(*Przepisanie wystąpienia warningów*)
VIS.uliWarningOccure.0:= TanksWarning[0].bWarning; 			AudiActiveWarningDescriptionIDtemp[0] := 25;
VIS.uliWarningOccure.1:= TanksWarning[1].bWarning; 			AudiActiveWarningDescriptionIDtemp[1] := 26;
VIS.uliWarningOccure.2:= BottleTransferWarning[0].bWarning; AudiActiveWarningDescriptionIDtemp[2] := 57;
VIS.uliWarningOccure.3:= GeneralWarning1[0].bWarning;		AudiActiveWarningDescriptionIDtemp[3] := 65;
VIS.uliWarningOccure.4:= WeightWarning[0].bWarning;	AudiActiveWarningDescriptionIDtemp[4] := 73;
VIS.uliWarningOccure.5:= BottleTransferWarning[1].bWarning;	AudiActiveWarningDescriptionIDtemp[5] := 58;
VIS.uliWarningOccure.6:= GeneralWarning1[0].bWarning;	AudiActiveWarningDescriptionIDtemp[6] := 65;
VIS.uliWarningOccure.7:= GeneralWarning1[1].bWarning;	AudiActiveWarningDescriptionIDtemp[7] := 66;
VIS.uliWarningOccure.8:= GeneralWarning1[2].bWarning;	AudiActiveWarningDescriptionIDtemp[8] := 67;
VIS.uliWarningOccure.9:= GeneralWarning1[3].bWarning;	AudiActiveWarningDescriptionIDtemp[9] := 68;
VIS.uliWarningOccure.10:=DispencersWarning[0].bWarning;	AudiActiveWarningDescriptionIDtemp[10] := 17;
VIS.uliWarningOccure.11:=DispencersWarning[1].bWarning;	AudiActiveWarningDescriptionIDtemp[11] := 18;
VIS.uliWarningOccure.12:=DispencersWarning[2].bWarning;	AudiActiveWarningDescriptionIDtemp[12] := 19;
VIS.uliWarningOccure.13:=DispencersWarning[3].bWarning;	AudiActiveWarningDescriptionIDtemp[13] := 20;
VIS.uliWarningOccure.14:=DispencersWarning[4].bWarning;	AudiActiveWarningDescriptionIDtemp[14] := 21;
VIS.uliWarningOccure.15:=ScrewersWarning[0].bWarning; 	AudiActiveWarningDescriptionIDtemp[15] := 49;
VIS.uliWarningOccure.16:=ScrewersWarning[1].bWarning;	AudiActiveWarningDescriptionIDtemp[16] := 50;
VIS.uliWarningOccure.17:=ScrewersWarning[2].bWarning;	AudiActiveWarningDescriptionIDtemp[17] := 51;
VIS.uliWarningOccure.18:=ScrewersWarning[3].bWarning;	AudiActiveWarningDescriptionIDtemp[18] := 52;
VIS.uliWarningOccure.19:=ScrewersWarning[4].bWarning;	AudiActiveWarningDescriptionIDtemp[19] := 53;
VIS.uliWarningOccure.20:=ScrewersWarning[5].bWarning;	AudiActiveWarningDescriptionIDtemp[20] := 54;
VIS.uliWarningOccure.21:=ScrewersWarning[6].bWarning;	AudiActiveWarningDescriptionIDtemp[21] := 55;
VIS.uliWarningOccure.22:=ScrewersWarning[7].bWarning;	AudiActiveWarningDescriptionIDtemp[22] := 56;
VIS.uliWarningOccure.23:=BottleFeederWarning[0].bWarning; 	AudiActiveWarningDescriptionIDtemp[23] := 1;
VIS.uliWarningOccure.24:=ExSensorWarning[1].bWarning;	AudiActiveWarningDescriptionIDtemp[24] := 90;
VIS.uliWarningOccure.25:=CapFeederWarning[0].bWarning;	AudiActiveWarningDescriptionIDtemp[25] := 33;
VIS.uliWarningOccure.26:=BottleFeederWarning[1].bWarning;	AudiActiveWarningDescriptionIDtemp[26] := 2;

VIS.uliWarningOccure.41:=BottleFeederWarning[2].bWarning;	AudiActiveWarningDescriptionIDtemp[41] := 3;
VIS.uliWarningOccure.42:=BottleFeederWarning[3].bWarning;	AudiActiveWarningDescriptionIDtemp[42] := 4;

VIS.uliWarningOccure.27:=CapSorterWarning[0].bWarning;	AudiActiveWarningDescriptionIDtemp[27] := 41;
VIS.uliWarningOccure.28:=CapSorterWarning[1].bWarning;	AudiActiveWarningDescriptionIDtemp[28] := 42;
VIS.uliWarningOccure.29:=CapSorterWarning[2].bWarning;	AudiActiveWarningDescriptionIDtemp[29] := 43;
VIS.uliWarningOccure.30:=CapSorterWarning[3].bWarning;	AudiActiveWarningDescriptionIDtemp[30] := 44;
VIS.uliWarningOccure.31:=CapSorterWarning[4].bWarning;	AudiActiveWarningDescriptionIDtemp[31] := 45;
VIS.uliWarningOccure.32:=CapSorterWarning[5].bWarning;	AudiActiveWarningDescriptionIDtemp[32] := 46;

VIS.uliWarningOccure.33:=BottleSorterWarning[0].bWarning;	AudiActiveWarningDescriptionIDtemp[33] := 9;
VIS.uliWarningOccure.34:=BottleSorterWarning[1].bWarning;	AudiActiveWarningDescriptionIDtemp[34] := 10;
VIS.uliWarningOccure.35:=BottleSorterWarning[2].bWarning;	AudiActiveWarningDescriptionIDtemp[35] := 11;
VIS.uliWarningOccure.36:=BottleSorterWarning[3].bWarning;	AudiActiveWarningDescriptionIDtemp[36] := 12;
VIS.uliWarningOccure.37:=BottleSorterWarning[4].bWarning;	AudiActiveWarningDescriptionIDtemp[37] := 13;
VIS.uliWarningOccure.38:=BottleSorterWarning[5].bWarning;	AudiActiveWarningDescriptionIDtemp[48] := 14;

VIS.uliWarningOccure.39:=LidFeederWarning[0].bWarning;	AudiActiveWarningDescriptionIDtemp[39] := 		81;
VIS.uliWarningOccure.40:=LidFeederWarning[1].bWarning;	AudiActiveWarningDescriptionIDtemp[40] := 		82;

(*Potwierdź wszystkie ostrzeżenia*)
IF VIS.bWarningAcknowledgeAll THEN
	VIS.uliWarningAcknowledge	:=	2#111111111111111111111111111111111111111111111111111111111;
	VIS.bWarningAcknowledgeAll	:= 	FALSE;
	iWarningAcknowledgeAll		:=	iWarningAcknowledgeAll	+	1;  // Sprawdzanie ile razy było wciśnięte
END_IF

(*Potwierdzenia*)
IF VIS.uliWarningAcknowledge.0 THEN TanksWarning[0].bAcknowledge					:=TRUE;	END_IF
IF VIS.uliWarningAcknowledge.1 THEN TanksWarning[1].bAcknowledge					:=TRUE; END_IF
IF VIS.uliWarningAcknowledge.2 THEN BottleTransferWarning[0].bAcknowledge			:=TRUE; END_IF
IF VIS.uliWarningAcknowledge.3 THEN GeneralWarning1[0].bAcknowledge					:=TRUE; END_IF
IF VIS.uliWarningAcknowledge.4 THEN WeightWarning[0].bAcknowledge					:=TRUE; END_IF
IF VIS.bBottleTransferLubricationReset THEN BottleTransferWarning[1].bAcknowledge	:=TRUE; END_IF
IF VIS.uliWarningAcknowledge.6 THEN GeneralWarning1[1].bAcknowledge					:=TRUE; END_IF
IF VIS.uliWarningAcknowledge.7 THEN GeneralWarning1[2].bAcknowledge					:=TRUE; END_IF
IF VIS.uliWarningAcknowledge.8 THEN GeneralWarning1[3].bAcknowledge					:=TRUE; END_IF
IF VIS.uliWarningAcknowledge.9 THEN GeneralWarning1[4].bAcknowledge					:=TRUE; END_IF
IF VIS.uliWarningAcknowledge.10 THEN DispencersWarning[0].bAcknowledge				:=TRUE; END_IF
IF VIS.uliWarningAcknowledge.11 THEN DispencersWarning[1].bAcknowledge				:=TRUE; END_IF
IF VIS.uliWarningAcknowledge.12 THEN DispencersWarning[2].bAcknowledge				:=TRUE; END_IF
IF VIS.uliWarningAcknowledge.13 THEN DispencersWarning[3].bAcknowledge				:=TRUE; END_IF
IF VIS.uliWarningAcknowledge.14 THEN DispencersWarning[4].bAcknowledge				:=TRUE; END_IF
IF VIS.uliWarningAcknowledge.15 THEN ScrewersWarning[0].bAcknowledge				:=TRUE; END_IF
IF VIS.uliWarningAcknowledge.16 THEN ScrewersWarning[1].bAcknowledge				:=TRUE; END_IF
IF VIS.uliWarningAcknowledge.17 THEN ScrewersWarning[2].bAcknowledge				:=TRUE; END_IF
IF VIS.uliWarningAcknowledge.18 THEN ScrewersWarning[3].bAcknowledge				:=TRUE; END_IF
IF VIS.uliWarningAcknowledge.19 THEN ScrewersWarning[4].bAcknowledge				:=TRUE; END_IF
IF VIS.uliWarningAcknowledge.20 THEN ScrewersWarning[5].bAcknowledge				:=TRUE; END_IF
IF VIS.uliWarningAcknowledge.21 THEN ScrewersWarning[6].bAcknowledge				:=TRUE; END_IF
IF VIS.uliWarningAcknowledge.22 THEN ScrewersWarning[7].bAcknowledge				:=TRUE; END_IF
IF VIS.uliWarningAcknowledge.23 THEN BottleFeederWarning[0].bAcknowledge			:=TRUE; END_IF
IF VIS.uliWarningAcknowledge.24 THEN ExSensorWarning[1].bAcknowledge				:=TRUE; END_IF
IF VIS.uliWarningAcknowledge.25 THEN CapFeederWarning[0].bAcknowledge				:=TRUE; END_IF
IF VIS.uliWarningAcknowledge.26 THEN BottleFeederWarning[1].bAcknowledge			:=TRUE; END_IF	

IF VIS.uliWarningAcknowledge.41 THEN BottleFeederWarning[2].bAcknowledge			:=TRUE; END_IF	
IF VIS.uliWarningAcknowledge.42 THEN BottleFeederWarning[3].bAcknowledge			:=TRUE; END_IF	

IF VIS.uliWarningAcknowledge.27 THEN CapSorterWarning[0].bAcknowledge				:=TRUE; END_IF	
IF VIS.uliWarningAcknowledge.28 THEN CapSorterWarning[1].bAcknowledge				:=TRUE; END_IF
IF VIS.uliWarningAcknowledge.29 THEN CapSorterWarning[2].bAcknowledge				:=TRUE; END_IF
IF VIS.uliWarningAcknowledge.30 THEN CapSorterWarning[3].bAcknowledge				:=TRUE; END_IF
IF VIS.uliWarningAcknowledge.31 THEN CapSorterWarning[4].bAcknowledge				:=TRUE; END_IF
IF VIS.uliWarningAcknowledge.32 THEN CapSorterWarning[5].bAcknowledge				:=TRUE; END_IF

IF VIS.uliWarningAcknowledge.33 THEN BottleSorterWarning[0].bAcknowledge			:=TRUE; END_IF	
IF VIS.uliWarningAcknowledge.34 THEN BottleSorterWarning[1].bAcknowledge			:=TRUE; END_IF
IF VIS.uliWarningAcknowledge.35 THEN BottleSorterWarning[2].bAcknowledge			:=TRUE; END_IF
IF VIS.uliWarningAcknowledge.36 THEN BottleSorterWarning[3].bAcknowledge			:=TRUE; END_IF
IF VIS.uliWarningAcknowledge.37 THEN BottleSorterWarning[4].bAcknowledge			:=TRUE; END_IF
IF VIS.uliWarningAcknowledge.38 THEN BottleSorterWarning[5].bAcknowledge			:=TRUE; END_IF

IF VIS.uliWarningAcknowledge.39 THEN LidFeederWarning[0].bAcknowledge				:=TRUE; END_IF
IF VIS.uliWarningAcknowledge.40 THEN LidFeederWarning[1].bAcknowledge				:=TRUE; END_IF
//41 i 42 zajete

(*Opisy*)
VIS.AsWarningDescription[0]:=TanksWarning[0].sDescription;
VIS.AsWarningDescription[1]:=TanksWarning[1].sDescription;
VIS.AsWarningDescription[2]:=BottleTransferWarning[0].sDescription;
VIS.AsWarningDescription[3]:=GeneralWarning1[0].sDescription;
VIS.AsWarningDescription[4]:=WeightWarning[0].sDescription;
VIS.AsWarningDescription[5]:=BottleTransferWarning[1].sDescription;
VIS.AsWarningDescription[6]:=GeneralWarning1[1].sDescription;
VIS.AsWarningDescription[7]:=GeneralWarning1[2].sDescription;
VIS.AsWarningDescription[8]:=GeneralWarning1[3].sDescription;
VIS.AsWarningDescription[9]:=GeneralWarning1[4].sDescription;
VIS.AsWarningDescription[10]:=DispencersWarning[0].sDescription;
VIS.AsWarningDescription[11]:=DispencersWarning[1].sDescription;
VIS.AsWarningDescription[12]:=DispencersWarning[2].sDescription;
VIS.AsWarningDescription[13]:=DispencersWarning[3].sDescription;
VIS.AsWarningDescription[14]:=DispencersWarning[4].sDescription;
VIS.AsWarningDescription[15]:=ScrewersWarning[0].sDescription;
VIS.AsWarningDescription[16]:=ScrewersWarning[1].sDescription;
VIS.AsWarningDescription[17]:=ScrewersWarning[2].sDescription;
VIS.AsWarningDescription[18]:=ScrewersWarning[3].sDescription;
VIS.AsWarningDescription[19]:=ScrewersWarning[4].sDescription;
VIS.AsWarningDescription[20]:=ScrewersWarning[5].sDescription;
VIS.AsWarningDescription[21]:=ScrewersWarning[6].sDescription;
VIS.AsWarningDescription[22]:=ScrewersWarning[7].sDescription;
VIS.AsWarningDescription[23]:=BottleFeederWarning[0].sDescription;     
VIS.AsWarningDescription[24]:=ExSensorWarning[1].sDescription;
VIS.AsWarningDescription[25]:=CapFeederWarning[0].sDescription;
VIS.AsWarningDescription[26]:=BottleFeederWarning[1].sDescription;

VIS.AsWarningDescription[41]:=BottleFeederWarning[2].sDescription;
VIS.AsWarningDescription[42]:=BottleFeederWarning[3].sDescription;

VIS.AsWarningDescription[27]:=CapSorterWarning[0].sDescription;
VIS.AsWarningDescription[28]:=CapSorterWarning[1].sDescription;
VIS.AsWarningDescription[29]:=CapSorterWarning[2].sDescription;
VIS.AsWarningDescription[30]:=CapSorterWarning[3].sDescription;
VIS.AsWarningDescription[31]:=CapSorterWarning[4].sDescription;
VIS.AsWarningDescription[32]:=CapSorterWarning[5].sDescription;

VIS.AsWarningDescription[33]:=BottleSorterWarning[0].sDescription;
VIS.AsWarningDescription[34]:=BottleSorterWarning[1].sDescription;
VIS.AsWarningDescription[35]:=BottleSorterWarning[2].sDescription;
VIS.AsWarningDescription[36]:=BottleSorterWarning[3].sDescription;
VIS.AsWarningDescription[37]:=BottleSorterWarning[4].sDescription;
VIS.AsWarningDescription[38]:=BottleSorterWarning[5].sDescription;

VIS.AsWarningDescription[39]:=LidFeederWarning[0].sDescription;
VIS.AsWarningDescription[40]:=LidFeederWarning[1].sDescription;
//41 i 42 zajete


(*SYGNALIZOWANIE WARNINGOW*)
tonSoftAlarm(IN:=bSoftAlarm, PT:=T#500MS);
rtWarningOccure0(CLK:=VIS.uliWarningOccure.0,Q=>);
rtWarningOccure1(CLK:=VIS.uliWarningOccure.1,Q=>);
rtWarningOccure2(CLK:=VIS.uliWarningOccure.2,Q=>);
rtWarningOccure3(CLK:=VIS.uliWarningOccure.3,Q=>);
rtWarningOccure4(CLK:=VIS.uliWarningOccure.4,Q=>);
rtWarningOccure5(CLK:=VIS.uliWarningOccure.5,Q=>);
rtWarningOccure6(CLK:=VIS.uliWarningOccure.6,Q=>);
rtWarningOccure7(CLK:=VIS.uliWarningOccure.7,Q=>);
rtWarningOccure8(CLK:=VIS.uliWarningOccure.8,Q=>);
rtWarningOccure9(CLK:=VIS.uliWarningOccure.9,Q=>);
rtWarningOccure10(CLK:=VIS.uliWarningOccure.10,Q=>);
rtWarningOccure11(CLK:=VIS.uliWarningOccure.11,Q=>);
rtWarningOccure12(CLK:=VIS.uliWarningOccure.12,Q=>);
rtWarningOccure13(CLK:=VIS.uliWarningOccure.13,Q=>);
rtWarningOccure14(CLK:=VIS.uliWarningOccure.14,Q=>);
rtWarningOccure15(CLK:=VIS.uliWarningOccure.15,Q=>);
rtWarningOccure16(CLK:=VIS.uliWarningOccure.16,Q=>);
rtWarningOccure17(CLK:=VIS.uliWarningOccure.17,Q=>);
rtWarningOccure18(CLK:=VIS.uliWarningOccure.18,Q=>);
rtWarningOccure19(CLK:=VIS.uliWarningOccure.19,Q=>);
rtWarningOccure20(CLK:=VIS.uliWarningOccure.20,Q=>);
rtWarningOccure21(CLK:=VIS.uliWarningOccure.21,Q=>);
rtWarningOccure22(CLK:=VIS.uliWarningOccure.22,Q=>);
rtWarningOccure23(CLK:=VIS.uliWarningOccure.23,Q=>);
rtWarningOccure24(CLK:=VIS.uliWarningOccure.24,Q=>);
rtWarningOccure25(CLK:=VIS.uliWarningOccure.25,Q=>);
rtWarningOccure26(CLK:=VIS.uliWarningOccure.26,Q=>);

rtWarningOccure41(CLK:=VIS.uliWarningOccure.41,Q=>);
rtWarningOccure42(CLK:=VIS.uliWarningOccure.42,Q=>);

rtWarningOccure27(CLK:=VIS.uliWarningOccure.27,Q=>);
rtWarningOccure28(CLK:=VIS.uliWarningOccure.28,Q=>);
rtWarningOccure29(CLK:=VIS.uliWarningOccure.29,Q=>);
rtWarningOccure30(CLK:=VIS.uliWarningOccure.30,Q=>);
rtWarningOccure31(CLK:=VIS.uliWarningOccure.31,Q=>);
rtWarningOccure32(CLK:=VIS.uliWarningOccure.32,Q=>);

rtWarningOccure33(CLK:=VIS.uliWarningOccure.33,Q=>);
rtWarningOccure34(CLK:=VIS.uliWarningOccure.34,Q=>);
rtWarningOccure35(CLK:=VIS.uliWarningOccure.35,Q=>);
rtWarningOccure36(CLK:=VIS.uliWarningOccure.36,Q=>);
rtWarningOccure37(CLK:=VIS.uliWarningOccure.37,Q=>);
rtWarningOccure38(CLK:=VIS.uliWarningOccure.38,Q=>);

rtWarningOccure39(CLK:=VIS.uliWarningOccure.39,Q=>);
rtWarningOccure40(CLK:=VIS.uliWarningOccure.40,Q=>);

IF	(rtWarningOccure0.Q AND NOT VIS.uliWarningAcknowledge.0) OR
	(rtWarningOccure1.Q AND NOT VIS.uliWarningAcknowledge.1) OR
	(rtWarningOccure2.Q AND NOT VIS.uliWarningAcknowledge.2) OR
	(rtWarningOccure3.Q AND NOT VIS.uliWarningAcknowledge.3) OR
	(rtWarningOccure4.Q AND NOT VIS.uliWarningAcknowledge.4) OR
	(rtWarningOccure5.Q AND NOT VIS.uliWarningAcknowledge.5) OR
	(rtWarningOccure6.Q AND NOT VIS.uliWarningAcknowledge.6) OR	
	(rtWarningOccure7.Q AND NOT VIS.uliWarningAcknowledge.7) OR	
	(rtWarningOccure8.Q AND NOT VIS.uliWarningAcknowledge.8) OR	
	(rtWarningOccure9.Q AND NOT VIS.uliWarningAcknowledge.9) OR	
	(rtWarningOccure10.Q AND NOT VIS.uliWarningAcknowledge.10) OR	
	(rtWarningOccure11.Q AND NOT VIS.uliWarningAcknowledge.11) OR	
	(rtWarningOccure12.Q AND NOT VIS.uliWarningAcknowledge.12) OR	
	(rtWarningOccure13.Q AND NOT VIS.uliWarningAcknowledge.13) OR	
	(rtWarningOccure14.Q AND NOT VIS.uliWarningAcknowledge.14) OR	
	(rtWarningOccure15.Q AND NOT VIS.uliWarningAcknowledge.15) OR	
	(rtWarningOccure16.Q AND NOT VIS.uliWarningAcknowledge.16) OR	
	(rtWarningOccure17.Q AND NOT VIS.uliWarningAcknowledge.17) OR	
	(rtWarningOccure18.Q AND NOT VIS.uliWarningAcknowledge.18) OR	
	(rtWarningOccure19.Q AND NOT VIS.uliWarningAcknowledge.19) OR	
	(rtWarningOccure20.Q AND NOT VIS.uliWarningAcknowledge.20) OR	
	(rtWarningOccure21.Q AND NOT VIS.uliWarningAcknowledge.21) OR	
	(rtWarningOccure22.Q AND NOT VIS.uliWarningAcknowledge.22) OR
	(rtWarningOccure23.Q AND NOT VIS.uliWarningAcknowledge.23) OR
	(rtWarningOccure24.Q AND NOT VIS.uliWarningAcknowledge.24) OR
	(rtWarningOccure25.Q AND NOT VIS.uliWarningAcknowledge.25) OR
	(rtWarningOccure26.Q AND NOT VIS.uliWarningAcknowledge.26) OR
	(rtWarningOccure41.Q AND NOT VIS.uliWarningAcknowledge.41) OR
	(rtWarningOccure42.Q AND NOT VIS.uliWarningAcknowledge.42) OR
	(rtWarningOccure27.Q AND NOT VIS.uliWarningAcknowledge.27) OR
	(rtWarningOccure28.Q AND NOT VIS.uliWarningAcknowledge.28) OR
	(rtWarningOccure29.Q AND NOT VIS.uliWarningAcknowledge.29) OR
	(rtWarningOccure30.Q AND NOT VIS.uliWarningAcknowledge.30) OR
	(rtWarningOccure31.Q AND NOT VIS.uliWarningAcknowledge.31) OR
	(rtWarningOccure32.Q AND NOT VIS.uliWarningAcknowledge.32) OR
	(rtWarningOccure33.Q AND NOT VIS.uliWarningAcknowledge.33) OR
	(rtWarningOccure34.Q AND NOT VIS.uliWarningAcknowledge.34) OR
	(rtWarningOccure35.Q AND NOT VIS.uliWarningAcknowledge.35) OR
	(rtWarningOccure36.Q AND NOT VIS.uliWarningAcknowledge.36) OR
	(rtWarningOccure37.Q AND NOT VIS.uliWarningAcknowledge.37) OR
	(rtWarningOccure38.Q AND NOT VIS.uliWarningAcknowledge.38) OR
	(rtWarningOccure39.Q AND NOT VIS.uliWarningAcknowledge.39) OR
	(rtWarningOccure40.Q AND NOT VIS.uliWarningAcknowledge.40) 
	
	
 THEN
	bSoftAlarm:=TRUE;
END_IF
IF tonSoftAlarm.Q THEN
	bSoftAlarm:=FALSE;
END_IF


(*Wykrywanie nowego ostrzezenia do wizualizacji*)
rtWarningNew ( CLK:= uliWarningAcknowledgeTemp	<> VIS.uliWarningOccure AND VIS.uliWarningOccure > 0);
uliWarningAcknowledgeTemp	:=	VIS.uliWarningOccure;
IF rtWarningNew.Q THEN
	VIS.bWarningNew	:=	TRUE;
END_IF
tonWarningNew (IN:= VIS.bWarningNew ,PT:=T#1S);
IF tonWarningNew.Q THEN
	VIS.bWarningNew	:=	FALSE;
END_IF
(*Koniec Wykrywanie nowego ostrzezenia do wizualizacji*)
END_ACTION

END_PROGRAM

// ---- POUs/P11_RollerScrewer.TcPOU
(*
Nazwa:			P11_RollerScrewer
Opis:			Stacja zakręcarki rolkowej
Wersja:			v0.1
Data:			2018-10-10
Autor:			DP
Urzadzenia:		
Konfiguracja:	
Info:

*)
PROGRAM P11_RollerScrewer
VAR_INPUT

END_VAR
VAR
	(*********Zakręcarka rolkowa******)
	fbRollerScrewer: FB_RollerScrewer;		// Blok sterowania zakręcarką rolkową
	eRollerScrewerState: 			E_Station;						// Stan zakręcarki
	eRollerScrewerRunningState: 	E_RollerScrewer;				// Stan zakręcarki
	fbRollerScrewerState: 			FB_State;
	
	(************Chwytak*************)	
	fbRollerScrewerCatchStation						: FB_CatchStation;		
	eRollerScrewerCatchState						: E_Station;            
	eRollerScrewerCatchRunningState					: E_CatchStationState;  
	fbRollerScrewerCatchState						: FB_State;
	
	(************Szlaban*************)		
	fbRollerScrewerGate								: FB_SpringGateV2;

	
	// WEJŚĆIA I WYJŚCIA SPRZĘTOWE
	IbRollerScrewerHeightEncoderSetCDone			AT %I*: BOOL;
	IudiRollerScrewerHeightEncoderCV          		AT %I*: UDINT;
	QbRollerScrewerHeightEncoderSetC 				AT %Q*: BOOL;
	QudiRollerScrewerHeightEncoderSetCV       		AT %Q*: UDINT;

	QbRollerScrewerCatchHeightUpCmd 				AT %Q*: BOOL; 		
	QbRollerScrewerCatchHeightDownCmd 				AT %Q*: BOOL; 		
	IbRollerScrewerCatchHeightEncoderSetCDone		AT %I*: BOOL;
	IudiRollerScrewerCatchHeightEncoderCV          	AT %I*: UDINT;
	QbRollerScrewerCatchHeightEncoderSetC 			AT %Q*: BOOL;
	QudiRollerScrewerCatchHeightEncoderSetCV       	AT %Q*: UDINT;

	QABPneumaticRollerScrewerValveCoils 			AT %Q* 	: ARRAY[1..5] OF BYTE;	
	IuiPneumaticRollerScrewerState					AT %I* 	: UINT;	


	IbRollerScrewerFuseFB1OK						AT %I*	:BOOL;		
	IbRollerScrewerFuseRollerScrewerOK				AT %I*	:BOOL;		
	IbRollerScrewerFuseRollerScrewerCatchOK			AT %I*	:BOOL;		
	IbRollerScrewerPowerSupplyOK					AT %I*	:BOOL;
	//GVL_IO_SAFETY.IbSafetyRelayRC40	 			AT %I*  :BOOL;	
	IbRollerScrewerDoors1Open 						AT %I*	:BOOL;		
	IbRollerScrewerCycleStartStopButton				AT %I*	:BOOL;	
	IbRollerScrewerCompressedAirOK 					AT %I*	:BOOL;		
	IbRollerScrewerUnPressedTopSensor 				AT %I*	:BOOL;	
	IbRollerScrewerRollsUnPressedSensor 			AT %I*	:BOOL; 

	IbRollerScrewerCatchSensorOpened				AT %I*	:BOOL; 
	IbRollerScrewerDoors2Open 						AT %I*	:BOOL;			
	IbRollerScrewerCapPuttedSensor 					AT %I*	:BOOL;	
	QbRollerScrewerGreenSignalizationLamp 			AT %Q* : BOOL;			
	QbRollerScrewerRedSignalizationLamp 			AT %Q* : BOOL;				
	QbRollerScrewerWhiteSignalizationLamp 			AT %Q* : BOOL;						
	QbRollerScrewerYellowSignalizationLamp 			AT %Q* : BOOL;							
	QbRollerScrewerHeightMotorUp 					AT %Q*: BOOL;		
	QbRollerScrewerHeightMotorDown 					AT %Q*: BOOL;			
	
	QbRollerScrewerGate								: BOOL; 	
	QbRollerScrewerPressingTopActuator				: BOOL; 	
	QbRollerScrewerPressingRollsActuator			: BOOL; 	
	QbRollerScrewerCatchActuator					: BOOL; 

	QnRollerScrewerFrontTorqueLimit 				AT %Q*: UINT; 
	QnRollerScrewerRearTorqueLimit 					AT %Q*: UINT; 
	IrRollerScrewerRearActualMotorTemperature 		AT %I*: REAL; 
	IrRollerScrewerFrontActualMotorTemperature 		AT %I*: REAL; 

	(*RFID*)
	//Przed
	bReadedCard 										: BOOL;				
	nReadedCard											: ULINT;	
	fbReader   											: FB_IfmIoLinkRfid;
	AusiReaderInputData  								AT %I* : ARRAY[0..27] OF USINT;
	IbReaderTagPresent									AT %I* : BOOL;
	IBReaderErrorValue									AT %I* : BYTE;
	IbReaderCmdEnd										AT %I* : BOOL;
	IBReaderDataCounterIn								AT %I* : BYTE;
	IbReaderCmdStartAck									AT %I* : BOOL;
	IbReaderCmdStart									AT %Q* : BOOL;
	IBReaderCmmandValue									AT %Q* : BYTE;
	IBReaderDataCounterOut								AT %Q* : BYTE;
	AusiReaderOutputData  								AT %Q* : ARRAY[0..27] OF USINT;	


	TimerRollerScrewerEnable: TOF;
	TimerRollerScrewerCatchEnable: TOF;
	tonLidPuttedCheckEnable: TON;	
	rtEnable: R_TRIG;	
	
	(*Wykres dozowania*)
	fbRollerScrewingChart: FB_WriteDataToArrayString;

	rtStartRollerScrewing: R_TRIG;
	lrRollerScrewerAxisStartPosition: LREAL;

	tonRollerScrewerCatchSensorOpened: TON;
	


END_VAR

aPowerSupply();
aButtons();
aPneumatics();
aRFID();
aRFID_FB();
aSafety();
aSignalization();
aLimits();
a1_Gate();
a1_GateTime();
a2_RollerScrewer();
aWarnings();

(*** SKALOWANIE WARTOŚCI ZAKRĘCANIA Z Nm na % ***)
(* Wersja w Nm fbRollerScrewer.iScrewerSetTorque 
:=LREAL_TO_INT( 
													(lrRollerScrewingTightTorque/(INT_TO_LREAL(iPackageCapDiameter)*0.0633))*100
												 );*)
												 
fbRollerScrewer.iScrewerSetTorque :=LREAL_TO_INT(lrRollerScrewingTightTorque);												 
(*** KONIEC SKALOWANIE WARTOŚCI ZAKRĘCANIA Z Nm na % ***)

(*SYMULACJA CZUJNIKÓW*)
tonRollerScrewerCatchSensorOpened(IN:=NOT QbRollerScrewerCatchActuator, PT:=T#10MS);//bylo 300


(* BAZOWANIE - ZMIAN*)
tonLidPuttedCheckEnable(IN:=fbRollerScrewer.bEnable,PT:=T#5S); (*Dodany ton bo Wizka zjebnie wgrywa zmienne, najpierw włacza Enabla a potem dopiero wybiera recepture*)
//rtEnable(CLK:=fbRollerScrewer.bEnable,Q=>);
rtEnable(CLK:=tonLidPuttedCheckEnable.Q,Q=>);
// IF rtEnable.Q AND eMachineState>=E_MachineState.eReady AND eMachineState<>E_MachineState.eHardError  THEN
// 	VIS.bRollerScrewerCatchHeightSet:=TRUE;
// 	//VIS.bRollerScrewerHeightSet:=TRUE;
// ELSIF fbRollerScrewer.eState=E_Station.eHomingDone OR eMachineState=E_MachineState.eHardError THEN
//  	VIS.bRollerScrewerHeightSet:=FALSE;
// ELSIF  fbRollerScrewerCatchStation.eState=E_Station.eHomingDone OR eMachineState=E_MachineState.eHardError THEN
// 	VIS.bRollerScrewerHeightSet:=TRUE; //Zmiana LU208
// 	VIS.bRollerScrewerCatchHeightSet:=FALSE;
// END_IF
(*KONIEC BAZOWANIE - ZMIANA*)


(********* GENEROWANIE STANU STACJI DO WIZKI**********)
// fbRollerScrewerState(
// 	eState:=eRollerScrewerState , 
// 	bRun:=bStartRollerScrewing OR VIS.bManualStartRollerScrew,	
// 	eRollerScrewerRunningState:=eRollerScrewerRunningState , 
// 	sStateDesc=> VIS.sRollerScrewerState,
// 	iState=>VIS.iRollerScrewerState);
//fbRollerScrewerCatchState(
//	eState:=eRollerScrewerCatchState , 
//	bRun:=bRollerScrewerCatch,	
//	eCatchRunningState:=eRollerScrewerCatchRunningState , 
//	sStateDesc=> VIS.sRollerScrewerCatchState,
//	iState=>VIS.iRollerScrewerCatchState);	
(***** KONIEC GENEROWANIE STANU STACJI DO WIZKI*******)

(*Opoznienie wyłączanie enabla*)
TimerRollerScrewerEnable 		(IN:=bRollerScrewerEnable  AND NOT bChangeover , PT:=T#2S);
TimerRollerScrewerCatchEnable 	(IN:=bRollerScrewerEnable  AND NOT bChangeover , PT:=T#4S);
{warning 'Zmienione włączenie/wyłączanie rolkowej do testów'}

(*Przypisywanie wartości*)
IF fbRollerScrewerCatchStation.lrHeightMotorCV+24 <= 65 THEN //Warrtość minimalna stacji zakrecarki rolkowej
	fbRollerScrewer.lrMinHeight := 60; //Warrtość minimalna stacji zakrecarki rolkowej
ELSE	//Jezeli ponad minimalną to minimalna jest wartościa chwytaka
	fbRollerScrewer.lrMinHeight:=fbRollerScrewerCatchStation.lrHeightMotorCV+10; 
END_IF

(********KASOWANIE ROZKAZÓW CYKLI*********)
IF fbRollerScrewer.bCycleDone AND bManualMode THEN
	VIS_RS.bRollerScrewerRun := FALSE;
END_IF
(*****KONIEC KASOWANIA ROZKAZÓW CYKLI*****)

ACTION a1_Gate:
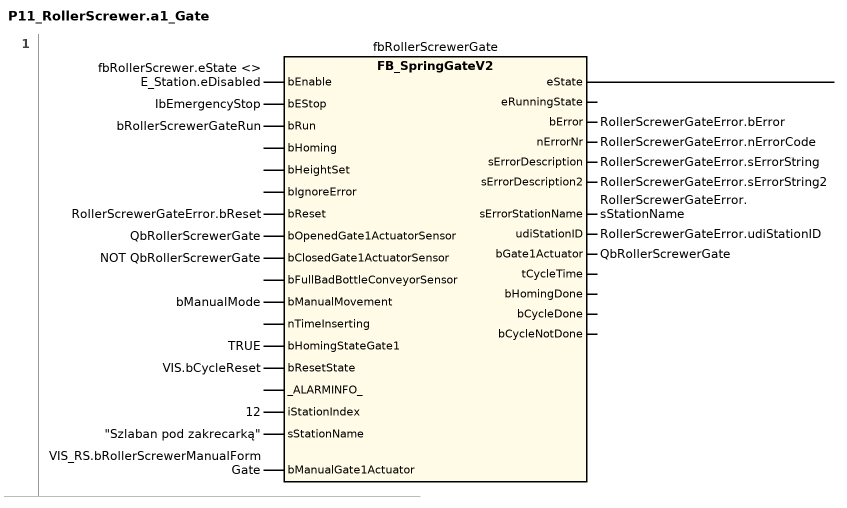
// NETWORK 1
fbRollerScrewerGate(
    bEnable := fbRollerScrewer.eState <> E_Station.eDisabled,
    bEStop := IbEmergencyStop,
    bRun := bRollerScrewerGateRun,
    bReset := RollerScrewerGateError.bReset,
    bOpenedGate1ActuatorSensor := QbRollerScrewerGate,
    bClosedGate1ActuatorSensor := NOT QbRollerScrewerGate,
    bManualMovement := bManualMode,
    bHomingStateGate1 := TRUE,
    bResetState := VIS.bCycleReset,
    iStationIndex := 12,
    sStationName := "Szlaban pod zakrecarką",
    bManualGate1Actuator := VIS_RS.bRollerScrewerManualFormGate,
    bError => RollerScrewerGateError.bError,
    nErrorNr => RollerScrewerGateError.nErrorCode,
    sErrorDescription => RollerScrewerGateError.sErrorString,
    sErrorDescription2 => RollerScrewerGateError.sErrorString2,
    sErrorStationName => RollerScrewerGateError.sStationName,
    udiStationID => RollerScrewerGateError.udiStationID,
    bGate1Actuator => QbRollerScrewerGate); // FB_SpringGateV2
END_ACTION

ACTION a1_GateTime:

fbRollerScrewerGate.nTimeInserting	:=	300;
END_ACTION

ACTION a2_RollerScrewer:
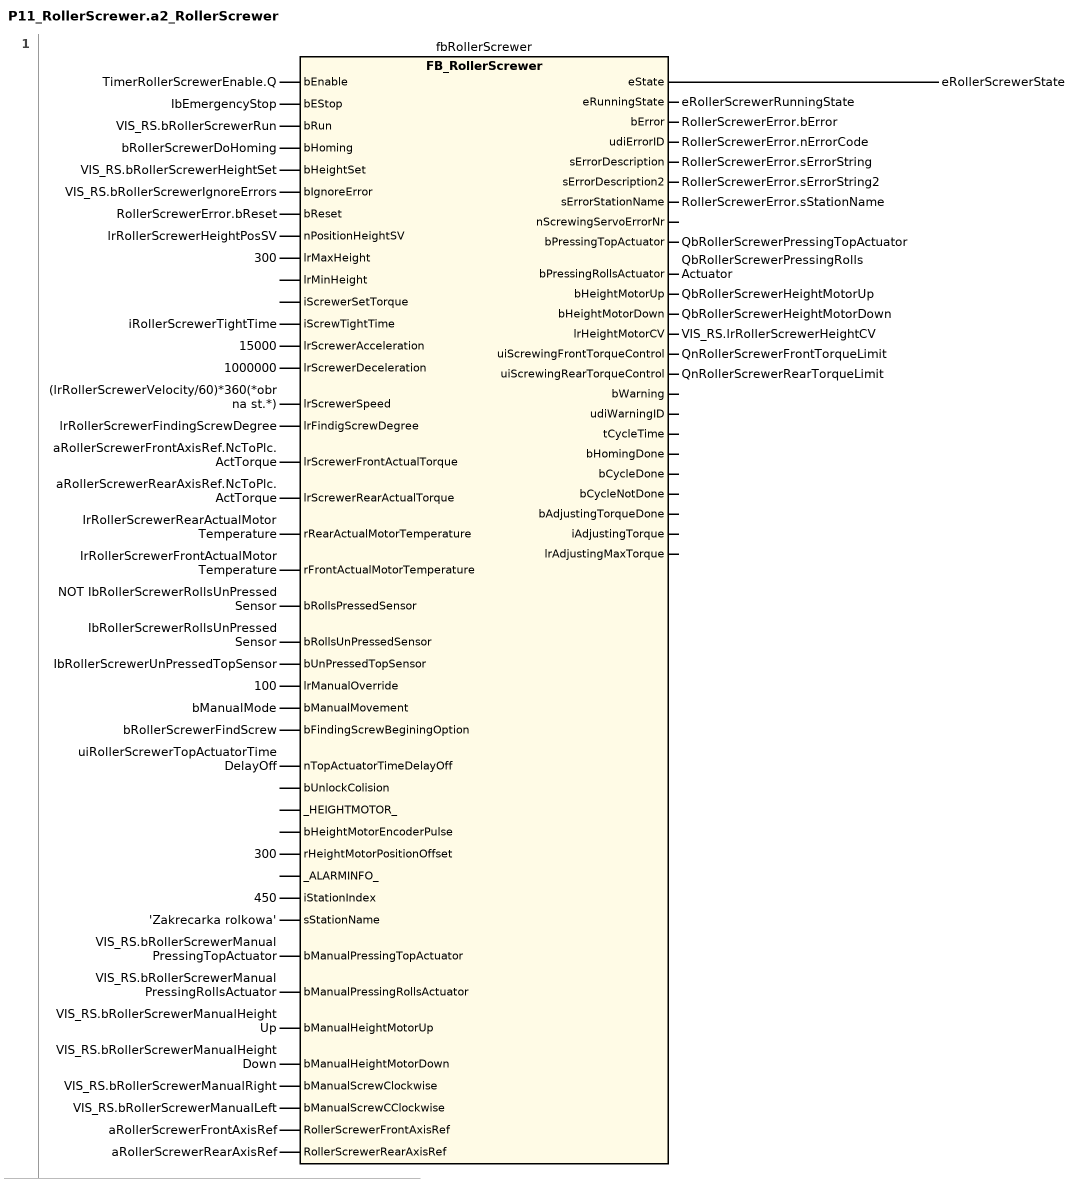
// NETWORK 1
fbRollerScrewer(
    bEnable := TimerRollerScrewerEnable.Q,
    bEStop := IbEmergencyStop,
    bRun := VIS_RS.bRollerScrewerRun,
    bHoming := bRollerScrewerDoHoming,
    bHeightSet := VIS_RS.bRollerScrewerHeightSet,
    bIgnoreError := VIS_RS.bRollerScrewerIgnoreErrors,
    bReset := RollerScrewerError.bReset,
    nPositionHeightSV := lrRollerScrewerHeightPosSV,
    lrMaxHeight := 300,
    iScrewTightTime := iRollerScrewerTightTime,
    lrScrewerAcceleration := 15000,
    lrScrewerDeceleration := 1000000,
    lrScrewerSpeed := (lrRollerScrewerVelocity/60)*360(*obr na st.*),
    lrFindigScrewDegree := lrRollerScrewerFindingScrewDegree,
    lrScrewerFrontActualTorque := aRollerScrewerFrontAxisRef.NcToPlc.ActTorque,
    lrScrewerRearActualTorque := aRollerScrewerRearAxisRef.NcToPlc.ActTorque,
    rRearActualMotorTemperature := IrRollerScrewerRearActualMotorTemperature,
    rFrontActualMotorTemperature := IrRollerScrewerFrontActualMotorTemperature,
    bRollsPressedSensor := NOT IbRollerScrewerRollsUnPressedSensor,
    bRollsUnPressedSensor := IbRollerScrewerRollsUnPressedSensor,
    bUnPressedTopSensor := IbRollerScrewerUnPressedTopSensor,
    lrManualOverride := 100,
    bManualMovement := bManualMode,
    bFindingScrewBeginingOption := bRollerScrewerFindScrew,
    nTopActuatorTimeDelayOff := uiRollerScrewerTopActuatorTimeDelayOff,
    rHeightMotorPositionOffset := 300,
    iStationIndex := 450,
    sStationName := 'Zakrecarka rolkowa',
    bManualPressingTopActuator := VIS_RS.bRollerScrewerManualPressingTopActuator,
    bManualPressingRollsActuator := VIS_RS.bRollerScrewerManualPressingRollsActuator,
    bManualHeightMotorUp := VIS_RS.bRollerScrewerManualHeightUp,
    bManualHeightMotorDown := VIS_RS.bRollerScrewerManualHeightDown,
    bManualScrewClockwise := VIS_RS.bRollerScrewerManualRight,
    bManualScrewCClockwise := VIS_RS.bRollerScrewerManualLeft,
    RollerScrewerFrontAxisRef := aRollerScrewerFrontAxisRef,
    RollerScrewerRearAxisRef := aRollerScrewerRearAxisRef,
    eRunningState => eRollerScrewerRunningState,
    bError => RollerScrewerError.bError,
    udiErrorID => RollerScrewerError.nErrorCode,
    sErrorDescription => RollerScrewerError.sErrorString,
    sErrorDescription2 => RollerScrewerError.sErrorString2,
    sErrorStationName => RollerScrewerError.sStationName,
    bPressingTopActuator => QbRollerScrewerPressingTopActuator,
    bPressingRollsActuator => QbRollerScrewerPressingRollsActuator,
    bHeightMotorUp => QbRollerScrewerHeightMotorUp,
    bHeightMotorDown => QbRollerScrewerHeightMotorDown,
    lrHeightMotorCV => VIS_RS.lrRollerScrewerHeightCV,
    uiScrewingFrontTorqueControl => QnRollerScrewerFrontTorqueLimit,
    uiScrewingRearTorqueControl => QnRollerScrewerRearTorqueLimit); // FB_RollerScrewer
eRollerScrewerState := fbRollerScrewer.eState;

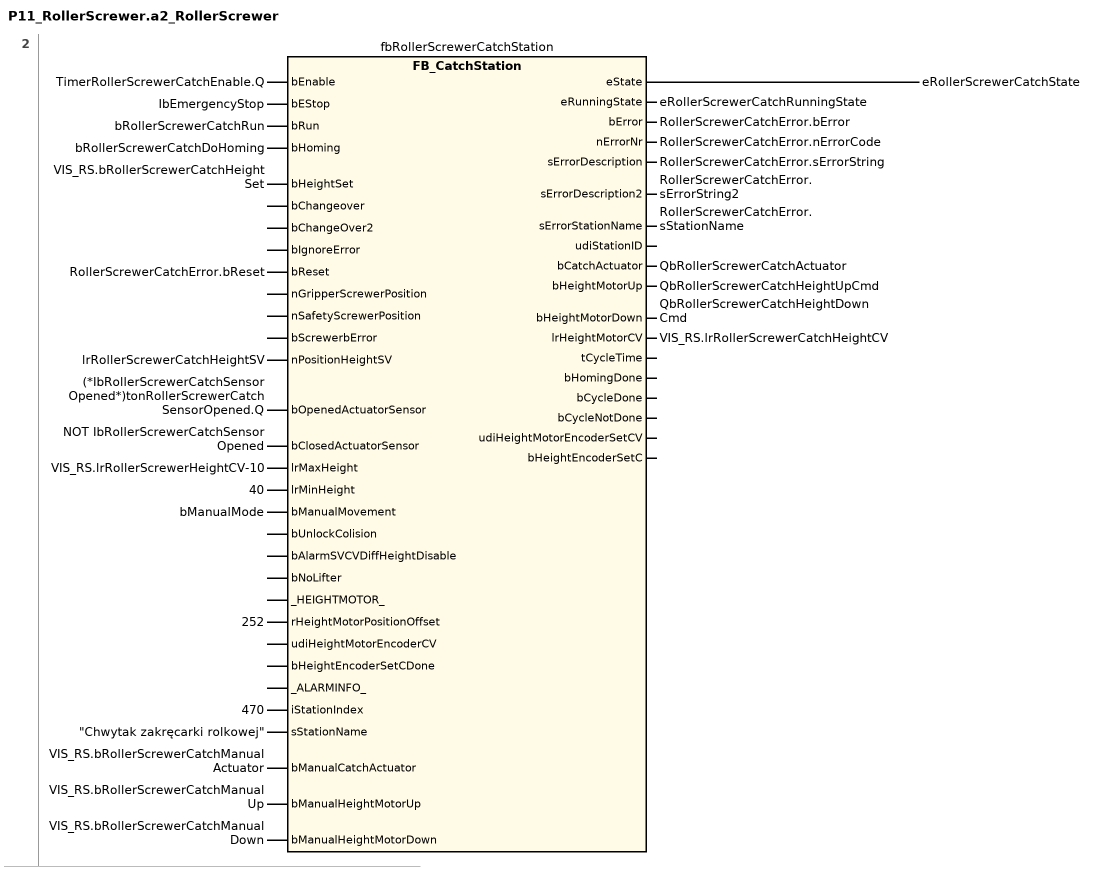
// NETWORK 2
fbRollerScrewerCatchStation(
    bEnable := TimerRollerScrewerCatchEnable.Q,
    bEStop := IbEmergencyStop,
    bRun := bRollerScrewerCatchRun,
    bHoming := bRollerScrewerCatchDoHoming,
    bHeightSet := VIS_RS.bRollerScrewerCatchHeightSet,
    bReset := RollerScrewerCatchError.bReset,
    nPositionHeightSV := lrRollerScrewerCatchHeightSV,
    bOpenedActuatorSensor := (*IbRollerScrewerCatchSensorOpened*)tonRollerScrewerCatchSensorOpened.Q,
    bClosedActuatorSensor := NOT IbRollerScrewerCatchSensorOpened,
    lrMaxHeight := VIS_RS.lrRollerScrewerHeightCV-10,
    lrMinHeight := 40,
    bManualMovement := bManualMode,
    rHeightMotorPositionOffset := 252,
    iStationIndex := 470,
    sStationName := "Chwytak zakręcarki rolkowej",
    bManualCatchActuator := VIS_RS.bRollerScrewerCatchManualActuator,
    bManualHeightMotorUp := VIS_RS.bRollerScrewerCatchManualUp,
    bManualHeightMotorDown := VIS_RS.bRollerScrewerCatchManualDown,
    eRunningState => eRollerScrewerCatchRunningState,
    bError => RollerScrewerCatchError.bError,
    nErrorNr => RollerScrewerCatchError.nErrorCode,
    sErrorDescription => RollerScrewerCatchError.sErrorString,
    sErrorDescription2 => RollerScrewerCatchError.sErrorString2,
    sErrorStationName => RollerScrewerCatchError.sStationName,
    bCatchActuator => QbRollerScrewerCatchActuator,
    bHeightMotorUp => QbRollerScrewerCatchHeightUpCmd,
    bHeightMotorDown => QbRollerScrewerCatchHeightDownCmd,
    lrHeightMotorCV => VIS_RS.lrRollerScrewerCatchHeightCV); // FB_CatchStation
eRollerScrewerCatchState := fbRollerScrewerCatchStation.eState;
END_ACTION

ACTION aButtons:

END_ACTION

ACTION aLimits:
(*
Nazwa:			aLimits
Opis:			Zabezpieczenia
Wersja:			v1.0
Data:			2023-11-24
Autor:			DP
Urzadzenia:		
Zmiany:	

Info:
*)

(**** Limity i zabezpieczenia***)
END_ACTION

ACTION aPneumatics:
// Do podpięcia według kolejności
QbRollerScrewerGate						;	
QbRollerScrewerPressingTopActuator		;
QbRollerScrewerPressingRollsActuator	;
QbRollerScrewerCatchActuator			;
;


(*************************** CapPusher EB1 **************************************)
// Wyspa 1 - dozowanie
IuiPneumaticRollerScrewerState;
QABPneumaticRollerScrewerValveCoils[1].0 := NOT QbRollerScrewerGate;
QABPneumaticRollerScrewerValveCoils[1].1 := QbRollerScrewerGate;
QABPneumaticRollerScrewerValveCoils[1].2 ;//
QABPneumaticRollerScrewerValveCoils[1].3 ;//
QABPneumaticRollerScrewerValveCoils[1].4 ;//
QABPneumaticRollerScrewerValveCoils[1].5 ;//
QABPneumaticRollerScrewerValveCoils[1].6 ;//
QABPneumaticRollerScrewerValveCoils[1].7 ;//
QABPneumaticRollerScrewerValveCoils[2].0 := QbRollerScrewerPressingTopActuator;			
QABPneumaticRollerScrewerValveCoils[2].1 ;
QABPneumaticRollerScrewerValveCoils[2].2 ;
QABPneumaticRollerScrewerValveCoils[2].3 ;
QABPneumaticRollerScrewerValveCoils[2].4 := QbRollerScrewerPressingRollsActuator;
QABPneumaticRollerScrewerValveCoils[2].5 ;
QABPneumaticRollerScrewerValveCoils[2].6 := QbRollerScrewerCatchActuator;
QABPneumaticRollerScrewerValveCoils[2].7 ;										                                                        
(*********************Koniec CapPusher EB1 **************************************)
END_ACTION

ACTION aPowerSupply:


	//Dodane do głwnych
	IbRollerScrewerFuseFB1OK				;
	IbRollerScrewerFuseRollerScrewerOK		;
	IbRollerScrewerFuseRollerScrewerCatchOK	;
	IbRollerScrewerPowerSupplyOK			;
END_ACTION

ACTION aRFID:
(*Przepisanie bity wykrycia karty*)
bReadedCard 		:= IbReaderTagPresent AND fbReader.bCodeReaded;
nReadedCard 		:= DINT_TO_ULINT(fbReader.diReadedCode);
END_ACTION

ACTION aRFID_FB:
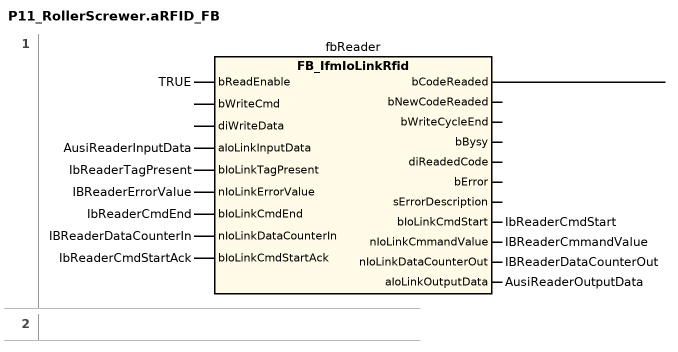
// NETWORK 1
fbReader(
    bReadEnable := TRUE,
    aIoLinkInputData := AusiReaderInputData,
    bIoLinkTagPresent := IbReaderTagPresent,
    nIoLinkErrorValue := IBReaderErrorValue,
    bIoLinkCmdEnd := IbReaderCmdEnd,
    nIoLinkDataCounterIn := IBReaderDataCounterIn,
    bIoLinkCmdStartAck := IbReaderCmdStartAck,
    bIoLinkCmdStart => IbReaderCmdStart,
    nIoLinkCmmandValue => IBReaderCmmandValue,
    nIoLinkDataCounterOut => IBReaderDataCounterOut,
    aIoLinkOutputData => AusiReaderOutputData); // FB_IfmIoLinkRfid

// NETWORK 2
END_ACTION

ACTION aRollerScrewerChartHMI:
(*Wykres zakręcarki rolkowej*)
rtStartRollerScrewing(CLK:=bStartRollerScrewing OR VIS.bManualStartRollerScrew, Q=>);
IF rtStartRollerScrewing.Q THEN (*Przy starcie zarkęcania, zapamiętywanie pozycji poczatkowej*)
	lrRollerScrewerAxisStartPosition := aRollerScrewerFrontAxisRef.NcToPlc.ActPos;
END_IF
 fbRollerScrewingChart(
	bWrite:= bStartRollerScrewing OR VIS.bManualStartRollerScrew, 
	nCycleTime:= 5, 
	lrData1:= aRollerScrewerFrontAxisRef.NcToPlc.ActPos - lrRollerScrewerAxisStartPosition, (*Zamiana st. na obr*)(*Odjęcie pozycji poczatkowej*) 
	lrData2:= aRollerScrewerFrontAxisRef.NcToPlc.ActTorque,// Wersja w Nm(aRollerScrewerFrontAxisRef.NcToPlc.ActTorque/100.0)*(INT_TO_LREAL(iPackageCapDiameter)*0.0633),  
	bData3:= QbRollerScrewerPressingRollsActuator, 
	bData4:= QbRollerScrewerPressingTopActuator,
	bData5:= FALSE,
	bData2B_ON:= FALSE,
	AsData=>VIS.AsChartRollerScrewing );
END_ACTION

ACTION aSafety:

// Dodać do P00_Alarms.aGeneralAlarms
	//IbCapPusherEmergencyStopButton0Pressed;
	//IbCapPusherEmergencyStopButton1Pressed;
	
(*
	IF IbCapPusherEmergencyStopButton0Pressed THEN
		GeneralAlarms.nErrorCode:=1;			
		GeneralAlarms.sErrorString:='Stop Awaryjny, sprawdź bezpieczeństwo, zresetuj przyciskiem na panelu | Naciśnięty przycisk awaryjny 1 na CapPusher';	
	ELSIF  IbCapPusherEmergencyStopButton1Pressed THEN
		GeneralAlarms.nErrorCode:=2;
		GeneralAlarms.sErrorString:='Stop Awaryjny, sprawdź bezpieczeństwo, zresetuj przyciskiem na panelu | Naciśnięty przycisk awaryjny 2 na CapPusher';	
*)	
	

// Dodać do miejsca gdzie są zamykane drzwi	
// lub zostawić tak jak jest
	IbRollerScrewerDoors1Open ;
	IbRollerScrewerDoors2Open ;
END_ACTION

ACTION aSignalization:
(*****Listwy LED*****)

QbRollerScrewerRedSignalizationLamp		:= INT_TO_BOOL(P00_Signalization.QiLineRedSignalizationLamp);
QbRollerScrewerGreenSignalizationLamp	:= INT_TO_BOOL(P00_Signalization.QiLineGreenSignalizationLamp);
QbRollerScrewerYellowSignalizationLamp	:= INT_TO_BOOL(P00_Signalization.QiLineBlueSignalizationLamp);
QbRollerScrewerWhiteSignalizationLamp ;

//QbCapPusherStartLamp	:= P00_Signalization.QbStartLamp;	   
//QbCapPusherResetLamp	:= P00_Signalization.QbResetLamp;
END_ACTION

ACTION aWarnings:
//Warning 0
//IF fbCapPusherFeeder.bWarning1 AND NOT CapSorterWarning[0].bWarning THEN
//	CapSorterWarning[0].bWarning										:=TRUE;
//	CapSorterWarning[0].udiWarningCode									:=41;
//	CapSorterWarning[0].sDescription									:='Sorter nasadek | Brak nasadek w zasobniku';
//ELSIF NOT fbCapPusherFeeder.bWarning1 THEN 
//	CapSorterWarning[0].bWarning										:=FALSE;
//	CapSorterWarning[0].bAcknowledge									:=FALSE;
//	VIS.uliWarningAcknowledge.27										:=FALSE;
//ELSIF CapSorterWarning[0].bAcknowledge THEN                               
//	CapSorterWarning[0].bAcknowledge									:=TRUE;
//END_IF
END_ACTION

END_PROGRAM

// ---- POUs/FB/FB_RollerScrewer.TcPOU
(*
Nazwa:			FB_RollerScrewer
Opis:			Zakręcarka rolkowa
Wersja:			v0.5
Data:			2020-03-16
Autor:			DP
Urzadzenia:		Serwo zakręcania, podnosnik JIESANG, rolki, docisk z góry
Konfiguracja:	
Info:  
- ZMIANA ESTOP - blad w trybie manualnym po ESTOPIE
- Dddano kasowanie ruchów w górę po błędzie
- Dodano opisy błędów serwa
- Dodano błędy od nastaw powyżej max i min (error 7 i 8)
- Zmiana Homingów według CatchStation
- zmiana momentu zacisniecia rolek
*)

FUNCTION_BLOCK FB_RollerScrewer
VAR_INPUT
	bEnable:BOOL;						//Zezowlenie na pracę zakręcarki rolkowej
	bEStop:BOOL;						//Stop awaryjny nieaktywny
	bRun:BOOL;							//Rozkaz zakręcania 
	bHoming:BOOL;						//Zezwolenie na wykonanie bazowania i pozycjonowania zakręcarki rolkowej
	bHeightSet:BOOL;					//Ustaw wysokość
	bIgnoreError:BOOL;					//Ignorowania błędów cyklu pracy
	bReset:BOOL;						//Reset błędu, jeśli w stanie "eError"
	nPositionHeightSV:LREAL;			//Wysokość zadana na której ma znajdować się zakręcarka rolkowa
	lrMaxHeight:LREAL;					//Maksymalna wysokość zakręcarki rolkowej
	lrMinHeight:LREAL;					//Minimalna wysokość zakręcarki rolkowej
	iScrewerSetTorque:INT;				//Zadany moment dokręcania [%]
	iScrewTightTime:INT;				//Czas przytrzymania po uzyskaniu momentu [ms] 
	lrScrewerAcceleration:LREAL;			//Przyspieszenie zakręcarki rolkowej
	lrScrewerDeceleration:LREAL;			//Opóźnienie zakręcarki rolkowej
	lrScrewerSpeed:LREAL;				//Prędkość zakręcarki rolkowej
	lrFindigScrewDegree:LREAL;			//Kąt wycofania zakręcarki rolkowej przy szukaniu gwintu
	lrScrewerFrontActualTorque:LREAL;			//Aktualny moment [%]
	lrScrewerRearActualTorque:LREAL;			//Aktualny moment [%]
	rRearActualMotorTemperature :REAL;	// Aktualna temperatura silnika tylniego
	rFrontActualMotorTemperature :REAL;	// Aktualna temperatura silnika tylniego
	bRollsPressedSensor: BOOL; 			// Wejście czujnika zaciśnięcie rolek zakręcarki
	bRollsUnPressedSensor: BOOL; 		// Wejście czujnika odpuszczenia rolek zakręcarki
	bUnPressedTopSensor: BOOL;			// Wejscie czujnika wycofania docisku górnego zakręcarki rolkowej
	lrManualOverride:LREAL;				// Procentowa redukcja prędkości wszystkich serw (Tylko w trybie manualnym)
	bManualMovement:BOOL; 			// Uruchomienie trybu ruchów ręcznych
	bFindingScrewBeginingOption:BOOL; 	//OPCJA. Szukaj początku gwintu nakrętki i opakowania. Zakręcarka napjpierw obraca się w lewo, a po znalezienu gwintu przystepuje do zakręcania;
	nTopActuatorTimeDelayOff:UINT;  	//czas po którym odpusczany jest docisk górny
	bUnlockColision:BOOL:=FALSE;		//Odblokowywanie możliwośći kolizji

	_HEIGHTMOTOR_ :BOOL;	
	bHeightMotorEncoderPulse :BOOL;			//Sygnał impulsów enkodera siłownika
	rHeightMotorPositionOffset :REAL;		//Wysokość bazowani podnośnika
	
	_ALARMINFO_ :BOOL;
	iStationIndex:UDINT;				//Numer stacji 
	sStationName:STRING;				//Nazwa stacji	
	
END_VAR
VAR_OUTPUT
	eState: E_Station;				// Stan zakręcarki rolkowej
	eRunningState:E_RollerScrewer;	// Stan zakręcarki	
	bError: BOOL;					// Błąd stacji
	udiErrorID: UDINT;				// Nr błędu zakręcarki rolkowej
	sErrorDescription:STRING(200);	// Opis błędu
	sErrorDescription2: STRING(200);// Opis błędu
	sErrorStationName: STRING;		// Nazwa stacj
	nScrewingServoErrorNr: UDINT;	// Nr błędu serwo zakręcarki
	bPressingTopActuator: BOOL; 	// Sterowanie zaworem dociskania nakrętki zaciskarki rolkowej od góry
	bPressingRollsActuator: BOOL; 	// Sterowanie zaworem dociskania rolek od boku
	bHeightMotorUp:BOOL;			// Sterowanie silnikiem podnośnika  - RUCH W GÓRĘ
	bHeightMotorDown:BOOL;			// Sterowanie silnikiem podnośnika  - RUCH W DÓŁ
	lrHeightMotorCV:LREAL;			// Aktualna pozycja podnośnika
	uiScrewingFrontTorqueControl:UINT;	// Kontola momentu zakręcania	
	uiScrewingRearTorqueControl:UINT;	// Kontola momentu zakręcania	

	bWarning: BOOL;
	udiWarningID: UDINT;
	tCycleTime:TIME;		
	bHomingDone:BOOL;				// Wymagane ponowne bazowanie (blad podczas bazowania lub stop awaryjny)
	bCycleDone:BOOL;
	bCycleNotDone:BOOL;		
	bAdjustingTorqueDone:BOOL;
	iAdjustingTorque:INT;
	lrAdjustingMaxTorque: LREAL;
END_VAR

VAR
	tonHeightNoChange: TON; // Timer wykrycia braku ruchu siłownika zmiany wysokości stacji
	nLastPositionHeightCV: LREAL;// Pozycja podnośnika w poprzednim cyklu programu
	tonErrorHeightChange: TON; // Timer błędu podnośnika
	rtEncoderHomed:R_TRIG;
	tonCycleTimer:TON;
	rtrigCycleTimerRead:R_TRIG;
	
	mcScrewerFrontMoveVelocity		:MC_MoveVelocity; 	// Ruch prędkościowy
	mcScrewerFrontHalt				:MC_HALT; 			// Zatrzymanie zakręcania
	mcScrewerFrontManualMove		:MC_JOG; 			// Blok obrotu ręcznego zakręcarką
	mcScrewerFrontStop				:MC_Stop; 			// Trwałe zatrzymywanie Serwo
	mcScrewerFrontPower				:MC_POWER; 			// Zasilanie napędu zakręcarki
	fbScrewerFrontHardReset			:FB_SoEReset;
	mcScrewerFrontSoftReset			:MC_Reset;
	mcScrewerFrontSetPosition		:MC_SetPosition;
	mcScrewerFrontMoveRelative		:MC_MoveRelative;

	mcScrewerRearMoveVelocity		:MC_MoveVelocity; 	// Ruch prędkościowy
	mcScrewerRearHalt				:MC_HALT; 			// Zatrzymanie zakręcania
	mcScrewerRearManualMove			:MC_JOG; 			// Blok obrotu ręcznego zakręcarką
	mcScrewerRearStop				:MC_Stop; 			// Trwałe zatrzymywanie Serwo
	mcScrewerRearPower				:MC_POWER; 			// Zasilanie napędu zakręcarki
	fbScrewerRearHardReset			:FB_SoEReset;
	mcScrewerRearSoftReset			:MC_Reset;
	mcScrewerRearSetPosition		:MC_SetPosition;
	mcScrewerRearMoveRelative		:MC_MoveRelative;
	
	bScrewFound: BOOL; //Zakręcarka znalazła początek gwintu
	nMaxTorque: LREAL; //Maksymalny moment podczas szukania poczatku gwintu
	nMinTorque: LREAL; // Najmniejszy moment podczas szukania poczatku gwintu

	tonTightScrewingTimer: TON; // Timer potwierdzenia dokręcenia nakrętki
	bScrewed: BOOL; // Nakrętka zakręcona

	tonTooLongScrewing: TON; // Błąd zbyt długiego zakręcania

	bScrewerFrontServoPower: BOOL; // Zmienna sterujaca zasilaniem serwo Zakręcark
	bScrewerRearServoPower: BOOL; // Zmienna sterujaca zasilaniem serwo Zakręcark

	// Za długie szukanie gwintu
	tonTooLongFinding: TON;
	tonPosDiffError	:TON;
	bStopped: BOOL;
	// Ustawianie pozycji napedu zakrecającego po zakręceniu nakrętki


	// Pozycja rozpoczęcia zakrecania
	lrStartScrewingPos: LREAL;
	
	// Ruch relatywny zakręcarki

	lrStartPositionScrewerFront: LREAL;
	lrStartPositionScrewerRear: LREAL;	
	tonPressingTopDelay: TON;
	tonPressingRollsDelay: TON;
	tonUpPressRollsDelay: TON;
	tonPressingRollsReliseDelay: TON;
	tonTopActuatorDelayOff: TON;
	tonPushingCapDelay: TON;
	tonRollsPressedDelay: TON;
	tofMotorUpPermition: TOF;
	tofMotorDownPermition: TOF;
	tonLimitPosMinReachedDelay: TON;
	tonLimitPosMaxReachedDelay: TON;
	tonMaxHeight: TON;

	bStateError: BOOL;

	//Podnośnik Jiesang	
	fbHeightMotorEncoder			:FB_JiesangActuatorEncoder;	// Blok enkodera podnośnika chwytaka stabilizującego pod zakręcarką	
	bHeightMotorEncoderCounterReset	:BOOL; 						// Sygnał resetu enkodera
	bHeightMotorEncoderHomed		:BOOL;						// Informacja od enkodera że jest zbazowany

	eLastState						:E_Station;			// Stan ogólny bloku
	eLastRunningState				:E_RollerScrewer;	// Stan podbloku
	eLastStateTemp					:E_Station;			// Stan ogólny bloku
	eLastRunningStateTemp			:E_RollerScrewer;	// Stan podbloku	
	sWarningDescription				:STRING;
	
	nCaseAdjustingTorque: INT;
	tonAdjustingTightScrewingTimer: TON;
	tonAdjustingGripperClose: TON;
	uiAdjustingScrewerTorqueControl: UINT;
	bAdjustingScrewed: BOOL;
	tonAdjustingCase40: TON;
	bAdjustingSetTorqueAchieved: BOOL;
	bAdjustingTorqueTooHigh: BOOL;
	bAdjustingTorqueTooLow: BOOL;
	lrMotorNominalTorque: LREAL;
	lrScrewerActualTorqueNm: LREAL;
	
	tonDelayServoOn			: TON;

	tonRearActualMotorTemperatureTooHigh: TON;
	tonFrontActualMotorTemperatureTooHigh: TON;
END_VAR

VAR_IN_OUT
	bManualPressingTopActuator		:BOOL;		// Sterowanie w trybie serwisowym zaworem dociskania nakrętki zaciskarki rolkowej od góry
	bManualPressingRollsActuator	:BOOL;		// Sterowanie w trybie serwisowym zaworem dociskania rolek od boku
	bManualHeightMotorUp			:BOOL;		// Ruch ręczny podnośnika stacji w górę
	bManualHeightMotorDown			:BOOL;		// Ruch ręczny podnośnika stacji w dół
	bManualScrewClockwise			:BOOL;		// Ruch ręczny zakręcarką w kierunku wskazówek zegara;
	bManualScrewCClockwise			:BOOL;		// Ruch ręczny zakręcarką w kierunku przeciwnym do wskazówek zegara;
	RollerScrewerFrontAxisRef		:AXIS_REF;	// Struktura sterowania NC dla serwa zakręcania
	RollerScrewerRearAxisRef		:AXIS_REF;	// Struktura sterowania NC dla serwa zakręcania	

END_VAR

(*Przepisywanie Homingu , rozdzielenie wyjść*)

HeightMotor();
ErrorHandling();
Control();
ServoFrontControlBlocks();
ServoRearControlBlocks();
Statistics();

(*Zapisywanie ostatniego stanu*)
IF eLastStateTemp<>eState THEN
	eLastState := eLastStateTemp;
END_IF
eLastStateTemp := eState;
IF eLastRunningStateTemp<>eRunningState THEN
	eLastRunningState := eLastRunningStateTemp;
END_IF
eLastRunningStateTemp := eRunningState;
(*Koniec Zapisywanie ostatniego stanu*)


nLastPositionHeightCV:=lrHeightMotorCV;

ACTION Control:
	(** TIMERY**)
	rtEncoderHomed				(CLK:= bHeightMotorEncoderHomed,Q=>);
	tonHeightNoChange			(IN:= ((bHeightMotorUp OR bHeightMotorDown) AND (nLastPositionHeightCV=lrHeightMotorCV)), PT:= T#1S); 
	tonLimitPosMinReachedDelay	(IN:= (lrHeightMotorCV<=lrMinHeight) AND eState=E_Station.eHoming,PT:= T#2S);
	tonLimitPosMaxReachedDelay	(IN:= (lrHeightMotorCV>=lrMaxHeight) AND eState=E_Station.eHoming,PT:= T#2S);

	tonPressingRollsReliseDelay(IN:= NOT bPressingRollsActuator AND NOT bPressingTopActuator, PT:= T#40MS);	
	tonTightScrewingTimer		(IN:= (eRunningState=E_RollerScrewer.eScrewing) AND 
								NOT tonTightScrewingTimer.Q AND mcScrewerFrontMoveVelocity.Execute AND mcScrewerRearMoveVelocity.Execute AND 
								((lrScrewerFrontActualTorque>=iScrewerSetTorque) OR (lrScrewerRearActualTorque>=iScrewerSetTorque)) AND 
								ABS(RollerScrewerFrontAxisRef.NcToPlc.PosDiff)>360 AND ABS(RollerScrewerRearAxisRef.NcToPlc.PosDiff)>360 
								AND NOT bScrewed ,PT:= INT_TO_TIME(iScrewTightTime));
	tonTopActuatorDelayOff		(IN:= bPressingTopActuator AND eRunningState=E_RollerScrewer.eScrewing, PT:= UINT_TO_TIME(nTopActuatorTimeDelayOff));	
	tonPushingCapDelay			(IN:= (eRunningState=E_RollerScrewer.ePushingCap) AND (NOT bUnPressedTopSensor OR  nTopActuatorTimeDelayOff=0), PT:= T#100MS);
	tonRollsPressedDelay		(IN:= (eRunningState=E_RollerScrewer.ePushingCap) AND NOT bRollsUnpressedSensor, PT:= T#0MS); //bylo 200

	tonDelayServoOn				(IN:=(eState = E_Station.ePreparingToReady), PT:=T#2S);
	
	(*****Wyłączenie enable*****)
	IF NOT bEnable THEN
		IF eState <> E_Station.eDisabled AND eState <> E_Station.ePreparingToDisable THEN
				eState 								:= E_Station.ePreparingToDisable; 
		END_IF	
	END_IF

	(*****Estop*****)
	IF NOT bEstop  THEN	
		IF eState <> E_Station.eAborted AND eState <> E_Station.eAborting AND eState <> E_Station.eDisabled THEN
				eState 								:= E_Station.eAborting; 
		END_IF
	END_IF

	
	CASE eState OF
	/////////////////////////////	
		E_Station.eDisabled: 						// Stan nieaktywnosci (Stacja wyłączona) 
		
			IF bEnable THEN
				eState 								:= E_Station.ePreparingToReady; 
			END_IF 
			
    /////////////////////////////	    
		E_Station.eAborted: 						// Stan bezpiecznego zatrzymania (po Abortingu) 

			IF bEStop THEN
				eState 								:= E_Station.ePreparingToReady;
			END_IF
			
	/////////////////////////////	
		E_Station.eAborting:                 		// Stan bezpiecznego zatrzymywania (po EStopie)
		
			bHeightMotorDown		:=	FALSE;
			bHeightMotorUp			:=	FALSE;	
		
			bPressingTopActuator					:= FALSE;
			bPressingRollsActuator					:= FALSE;

			mcScrewerFrontPower.Override			:= 100;
			mcScrewerFrontStop.Execute				:= NOT bStopped;
			mcScrewerFrontMoveVelocity.Execute		:= FALSE;
			mcScrewerFrontManualMove.JogBackwards	:= FALSE;
			mcScrewerFrontManualMove.JogForward		:= FALSE;
			
			mcScrewerRearPower.Override				:= 100;
			mcScrewerRearStop.Execute				:= NOT bStopped;
			mcScrewerRearMoveVelocity.Execute		:= FALSE;
			mcScrewerRearManualMove.JogBackwards	:= FALSE;
			mcScrewerRearManualMove.JogForward		:= FALSE;
			
			IF ((mcScrewerFrontStop.Done OR NOT bScrewerFrontServoPower) AND (mcScrewerRearStop.Done OR NOT bScrewerRearServoPower)) OR bStopped THEN
				bStopped							:= FALSE;
				bScrewerFrontServoPower				:= FALSE;
				mcScrewerFrontStop.Execute			:= FALSE;
				bScrewerRearServoPower				:= FALSE;
				mcScrewerRearStop.Execute			:= FALSE;
				eState								:= E_Station.eAborted; 
				eRunningState						:= E_RollerScrewer.eReady;
			END_IF		
			
			
	/////////////////////////////			
		E_Station.eError:                 	 		// Stan błędu 	
				
			IF bReset THEN
				eState 								:= E_Station.eResetting;
			ELSE
				mcScrewerFrontSoftReset				(Execute:= FALSE,Axis:= RollerScrewerFrontAxisRef);	
				mcScrewerRearSoftReset				(Execute:= FALSE,Axis:= RollerScrewerRearAxisRef);	
			END_IF
			
	/////////////////////////////
		E_Station.eResetting:						// Stan resetowania bledu (po Errorze)
			
			//Procedura obsługi resetu w zależności od błędu
			CASE udiErrorID-iStationIndex OF
		
				//Error 1 - ZA DŁUGIE ZAKRĘCANIE	
				1:
					IF tonPressingRollsReliseDelay.Q AND RollerScrewerFrontAxisRef.Status.StandStill AND RollerScrewerRearAxisRef.Status.StandStill THEN
						;
						udiErrorID					:= 0;
						sErrorDescription			:= '';	
						bError 						:= FALSE;	
					END_IF
					
				//Error 2,4,5,6,7,8	
				2,4,5,6,7,8:   
					 bError 						:= FALSE;
					 udiErrorID						:= 0;
					 sErrorDescription				:= '';		
			
				//Error 3 - BŁĄD SERWA ZAKRĘCANIA
				3:	
					//fbScrewerHardReset			(Execute:= NOT mcHeightMoveAbsolute.Execute,Axis:= ScrewingAxisRef);
					mcScrewerFrontSoftReset			(Execute:= TRUE,Axis:= RollerScrewerFrontAxisRef);
					mcScrewerRearSoftReset			(Execute:= TRUE,Axis:= RollerScrewerRearAxisRef);
					IF NOT fbScrewerFrontHardReset.Busy AND NOT mcScrewerFrontSoftReset.Busy AND mcScrewerFrontPower.Status AND NOT RollerScrewerFrontAxisRef.Status.Error
					AND NOT fbScrewerRearHardReset.Busy AND NOT mcScrewerRearSoftReset.Busy AND mcScrewerRearPower.Status AND NOT RollerScrewerRearAxisRef.Status.Error  THEN
						fbScrewerFrontHardReset		(Execute:= FALSE,Axis:= RollerScrewerFrontAxisRef);
						fbScrewerRearHardReset		(Execute:= FALSE,Axis:= RollerScrewerRearAxisRef);
						mcScrewerFrontSoftReset		(Execute:= FALSE,Axis:= RollerScrewerFrontAxisRef);
						mcScrewerRearSoftReset		(Execute:= FALSE,Axis:= RollerScrewerRearAxisRef);
						bError 						:= FALSE;
						udiErrorID					:= 0;
						nScrewingServoErrorNr		:= 0;
						mcScrewerFrontPower.Override:= 100;
						mcScrewerRearPower.Override	:= 100;
						eState						:= E_Station.eReady;
						sErrorDescription			:= '';	
			
					ELSIF NOT fbScrewerFrontHardReset.Busy AND NOT mcScrewerFrontSoftReset.Busy AND NOT mcScrewerFrontPower.Status AND NOT bScrewerFrontServoPower AND NOT RollerScrewerFrontAxisRef.Status.Error
						AND NOT fbScrewerRearHardReset.Busy AND NOT mcScrewerRearSoftReset.Busy AND NOT mcScrewerRearPower.Status AND NOT bScrewerRearServoPower AND NOT RollerScrewerRearAxisRef.Status.Error THEN
						//fbScrewerHardReset(Execute:= FALSE,Axis:= ScrewingAxisRef);
						mcScrewerFrontSoftReset		(Execute:= FALSE,Axis:= RollerScrewerFrontAxisRef);
						mcScrewerRearSoftReset		(Execute:= FALSE,Axis:= RollerScrewerRearAxisRef);
						udiErrorID					:= 0;
						nScrewingServoErrorNr		:= 0;
						mcScrewerFrontPower.Override:= 100;
						mcScrewerRearPower.Override	:= 100;
						bError 						:= FALSE;
						sErrorDescription			:= '';
					END_IF		
					
			END_CASE	
			
			IF NOT bError THEN
				udiErrorID 							:= 	0;
   				sErrorDescription 					:= 	'';
	                                				
				eState 								:= 	E_Station.ePreparingToReady;
				mcScrewerFrontStop.Execute			:= FALSE;    
				mcScrewerRearStop.Execute			:= FALSE; 
			ELSE                    	
				eState 								:= 	E_Station.eError;
			END_IF
        
	/////////////////////////////
		E_Station.eManualMovement:     				// Stan ruchów manualnych  
       
			ManualMovements();
			//Wyjście z trybu serwisowego
			IF NOT bManualMovement THEN
				bManualPressingTopActuator			:= 	FALSE;
				bManualPressingRollsActuator		:= 	FALSE;
				bHeightMotorUp						:= 	FALSE;
				bHeightMotorDown					:= 	FALSE;
				mcScrewerFrontPower.Override			:= 	100;
				mcScrewerRearPower.Override			:= 	100;
				eState								:= 	E_Station.eReady;
			END_IF

	/////////////////////////////
		E_Station.eHoming:							// Stan bazowania 

			Homing();
			IF NOT bHoming AND NOT bHeightSet THEN
			   eState								:= 	E_Station.ePreparingToReady;
			   bHeightMotorUp						:= 	FALSE;
				bHeightMotorDown					:= 	FALSE;
			END_IF		
			
	/////////////////////////////
		E_Station.eHomingDone:                  	// Stan wykonania bazowania 

			bHeightMotorDown						:= 	FALSE;
			bHeightMotorUp							:= 	FALSE;
			bHeightMotorEncoderCounterReset			:= 	FALSE;
			bHomingDone								:= 	TRUE;
			IF NOT bHoming AND NOT bHeightSet THEN
			   	eState								:= 	E_Station.eReady;
			END_IF
			
	/////////////////////////////
		E_Station.ePreparingToReady:            	// Stan przygotowywania do gotowosci (zawsze przed Ready)  
	
			IF tonDelayServoOn.Q THEN
				bScrewerFrontServoPower				:= 	TRUE;
				bScrewerRearServoPower				:= 	TRUE;
			END_IF	

				
			bPressingTopActuator					:= 	FALSE;
			bPressingRollsActuator					:= 	FALSE;
			IF mcScrewerFrontPower.Status AND mcScrewerRearPower.Status THEN  	
				eState								:= 	E_Station.eReady;
				eRunningState						:= 	E_RollerScrewer.eReady;
			END_IF                              	
         	IF bIgnoreError THEN                	
				eState								:= 	E_Station.eReady;
				eRunningState						:= 	E_RollerScrewer.eReady;
			END_IF
	
	/////////////////////////////
		E_Station.ePreparingToDisable:         	 	// Stan przygotowywania do nieaktywnosci (po wyłączeniu Enable) 
  
			bScrewerFrontServoPower					:= 	TRUE;
			bScrewerRearServoPower					:= 	TRUE;

			
			bPressingTopActuator					:= 	FALSE;
			bPressingRollsActuator					:= 	FALSE;
			                        				
			bHeightMotorUp							:= 	TRUE;
			bHeightMotorDown						:= 	FALSE;
			IF tonHeightNoChange.Q THEN	
				bHeightMotorUp:= FALSE;
				IF  mcScrewerFrontPower.Status THEN
					bScrewerFrontServoPower			:= 	FALSE; //LU205
					bScrewerRearServoPower			:= 	FALSE;;//LU205
					eState							:= 	E_Station.eDisabled;
					eRunningState					:= 	E_RollerScrewer.eReady;
				END_IF
			END_IF				
         	IF bIgnoreError THEN
				bHeightMotorUp						:= 	FALSE;
				eState								:= 	E_Station.eDisabled;
				eRunningState						:= 	E_RollerScrewer.eReady;
			END_IF
			
	/////////////////////////////
		E_Station.eReady:							// Stan gotowosci 
		
			mcScrewerFrontStop.Execute:= FALSE;
		
			IF bRun AND NOT bCycleDone AND NOT bCycleNotDone THEN
				eState 								:= E_Station.eStarting; 
			END_IF
			IF bHoming OR bHeightSet THEN
				eState 								:= E_Station.eHoming; 
			END_IF
			IF bManualMovement THEN
				//Jeśli przejście w tryb ruchów manualnych przepisz wszystkie stany siłowników sterowanych przez moduł
				//aby zapobiec ewentualnym kolizjom po wejściu w tryb serwisowy
				bManualPressingTopActuator			:= 	bPressingTopActuator;
				bManualPressingRollsActuator		:= 	bPressingRollsActuator;
				bManualHeightMotorUp				:= 	bHeightMotorUp;
				bManualHeightMotorDown				:= 	bHeightMotorDown;
				mcScrewerFrontStop.Execute			:= 	FALSE;
				mcScrewerRearStop.Execute			:= 	FALSE;
				eState 								:= 	E_Station.eManualMovement; 
			END_IF
			IF NOT bRun THEN
				bCycleDone 							:= FALSE;
				bCycleNotDone 						:= FALSE;	
				bWarning							:= FALSE;	
			END_IF      

			bStopped								:= FALSE;
			mcScrewerFrontStop.Execute				:= FALSE;    
			mcScrewerRearStop.Execute				:= FALSE;                   			
			
	/////////////////////////////
		E_Station.eStopping:					// Stan zatrzymywania 
			
			Running();

			bPressingTopActuator					:= 	FALSE;
			bPressingRollsActuator					:= 	FALSE;
			
			mcScrewerFrontHalt.Execute				:= 	FALSE;			
			mcScrewerFrontStop.Execute				:= 	NOT bStopped;
			mcScrewerFrontMoveRelative.Execute		:= 	FALSE;
			mcScrewerFrontMoveVelocity.Execute		:= 	FALSE;
			uiScrewingFrontTorqueControl			:= 	0; // bylo 6000	
			mcScrewerFrontSoftReset					(Axis:= RollerScrewerFrontAxisRef, Execute:= TRUE);

			mcScrewerRearHalt.Execute				:= 	FALSE;			
			mcScrewerRearStop.Execute				:= 	NOT bStopped;
			mcScrewerRearMoveRelative.Execute		:= 	FALSE;
			mcScrewerRearMoveVelocity.Execute		:= 	FALSE;
			uiScrewingRearTorqueControl				:= 	0; // bylo 6000	
			mcScrewerRearSoftReset					(Axis:= RollerScrewerRearAxisRef, Execute:= TRUE);
			
			IF  (mcScrewerFrontStop.Done OR mcScrewerFrontStop.CommandAborted) AND 
				(mcScrewerRearStop.Done OR mcScrewerRearStop.CommandAborted) 
				THEN
				mcScrewerFrontStop.Execute			:= 	FALSE;
				mcScrewerRearStop.Execute			:= 	FALSE;
				bStopped							:= 	FALSE;
				eState 								:= 	E_Station.eReady;
			END_IF
		
		
	/////////////////////////////
		E_Station.eStarting:                  	// Stan uruchamiania (po Ready)
		
			eState									 := E_Station.eRunning; 
			
	/////////////////////////////
		E_Station.eRunning:               		// Stan wykonywania cyklu (po Startingu), w tym stanie osobny
 
			Running();
			IF NOT bRun THEN					(*Przerywanie cyklu*)
				eState 				 				:= E_Station.eStopping;	
			END_IF
			IF bCycleDone OR bCycleNotDone THEN (*Cykl zakończony*)
				eState 								 := E_Station.eReady;
			END_IF	
			
			
	/////////////////////////////		
	END_CASE
END_ACTION

ACTION ErrorHandling:
//OBSŁUGA BŁĘDÓW ZAKRĘCARKI ROLKOWEJ

RollerScrewerFrontAxisRef.ReadStatus();


//**********************LISTA BŁĘDÓW******************************
bStateError:= (eState=E_Station.eError) OR (eState=E_Station.eResetting) OR bIgnoreError;

IF bEnable THEN
	
	//Error 1 - ZA DŁUGIE ZAKRĘCANIE
	tonTooLongScrewing(IN:=(eRunningState=E_RollerScrewer.eScrewing),PT:=T#2S);
	tonTooLongFinding(IN:=(eRunningState=E_RollerScrewer.eFindingScrew),PT:=T#1S500MS);
	tonPosDiffError(IN:=((ABS(RollerScrewerFrontAxisRef.NcToPlc.ActPos-lrStartPositionScrewerFront)>=3080) OR ABS(RollerScrewerRearAxisRef.NcToPlc.ActPos-lrStartPositionScrewerRear)>=3080)  AND eRunningState=E_RollerScrewer.eScrewing,PT:=T#1MS);
	IF (tonTooLongScrewing.Q OR tonTooLongFinding.Q OR tonPosDiffError.Q) AND NOT bStateError THEN
		bHeightMotorUp:=FALSE;
		bHeightMotorDown:=FALSE;
		bStopped:=FALSE;
		bPressingTopActuator:=FALSE;
		bPressingRollsActuator:=FALSE;
		mcScrewerFrontMoveVelocity.Execute:=FALSE;
		mcScrewerFrontHalt.Execute:=FALSE;
		mcScrewerRearMoveVelocity.Execute:=FALSE;
		mcScrewerRearHalt.Execute:=FALSE;
		eState	:= E_Station.eStopping; 
		eRunningState	:=	E_RollerScrewer.eNotDone;
		bWarning:=TRUE;
		udiWarningID := 1;
		udiErrorID := 1;
		udiErrorID := udiErrorID+iStationIndex;
		sWarningDescription:='Przekroczenie czasu zakręcania - zmień ustawienia zakręcania';	
		(*Kasownie momentu po zakręceniu*)		
		uiScrewingFrontTorqueControl:=0; // bylo 6000
		uiScrewingRearTorqueControl:=0; // bylo 6000
		mcScrewerFrontSoftReset(Axis:=RollerScrewerFrontAxisRef, Execute:= TRUE);
		mcScrewerRearSoftReset(Axis:=RollerScrewerRearAxisRef, Execute:= TRUE);
	END_IF
	
	//Error 2 - podnośnik nie porusza się pomimo wysterowania 
	tonErrorHeightChange(IN:=(bHeightMotorUp OR bHeightMotorDown) AND nLastPositionHeightCV=lrHeightMotorCV, PT:=T#3S);
	IF tonErrorHeightChange.Q AND NOT bStateError THEN
		bHeightMotorUp:=FALSE;
		bHeightMotorDown:=FALSE;
		bError := TRUE;
		udiErrorID:=2;
		udiErrorID := udiErrorID+iStationIndex;	
		sErrorDescription:='Blokada podnośnika lub brak zasilania - sprawdź czujnik lub odblokuj mechanicznie';	
	END_IF
	
	//Error 3 - BŁĄD SERWA ZAKRĘCAJĄCEGO
	IF RollerScrewerFrontAxisRef.Status.Error OR mcScrewerFrontStop.Error OR RollerScrewerRearAxisRef.Status.Error OR mcScrewerRearStop.Error AND NOT bStateError THEN
		bHeightMotorUp:=FALSE;
		bHeightMotorDown:=FALSE;
		bStopped:=FALSE;
		bError := TRUE;
		udiErrorID:=3;
		udiErrorID := udiErrorID+iStationIndex;	
		nScrewingServoErrorNr:=RollerScrewerFrontAxisRef.Status.ErrorID;
		sErrorDescription:='Błąd napędu zakręcającego. Błąd NC:';
		sErrorDescription2:=F_AxErrMsg(nScrewingServoErrorNr);
	END_IF;
	
	//Error 4 - BLAD DOCISKU NAKRĘTKI OD GÓRY ZAKRECARKI
	tonPressingTopDelay(IN:=(NOT bPressingTopActuator AND NOT bUnPressedTopSensor),PT:=T#1S);
	IF tonPressingTopDelay.Q AND NOT bStateError THEN
		bHeightMotorUp:=FALSE;
		bHeightMotorDown:=FALSE;
		bPressingTopActuator:=FALSE;
		bError := TRUE;
		udiErrorID:=4;
		udiErrorID := udiErrorID+iStationIndex;			
		sErrorDescription:='Błąd docisku nakrętki od góry - sprawdź czujnik ';
	END_IF;
	
	//Error 5 - BLAD DOCISKU ROLEK DOCISKAJĄCYCH ZAKRECARKI
	tonPressingRollsDelay(IN:=(bPressingRollsActuator AND NOT bRollsPressedSensor),PT:=T#1S);
	IF tonPressingRollsDelay.Q AND NOT bStateError THEN
		bHeightMotorUp:=FALSE;
		bHeightMotorDown:=FALSE;
		bPressingRollsActuator:=FALSE;
		bError := TRUE;
		udiErrorID:=5;
		udiErrorID := udiErrorID+iStationIndex;			
		sErrorDescription:='Błąd docisku rolek - sprawdź czujnik';
	END_IF;
	
	//Error 6 - BLAD ODPUSZCZENIA ROLEK DOCISKAJĄCYCH ZAKRECARKI
	tonUpPressRollsDelay(IN:=(NOT bPressingRollsActuator AND NOT bRollsUnPressedSensor),PT:=T#1S);
	IF tonUpPressRollsDelay.Q AND NOT bStateError  THEN
		bHeightMotorUp:=FALSE;
		bHeightMotorDown:=FALSE;
		bPressingRollsActuator:=FALSE;
		bError := TRUE;
		udiErrorID:=6;
		udiErrorID := udiErrorID+iStationIndex;			
		sErrorDescription:='Błąd odocisku rolek - sprawdź czujnik';
	END_IF;
	
	//Error 7 - Bład nastaw max
	tonMaxHeight(IN:=nPositionHeightSV>lrMaxHeight AND NOT bHomingDone AND eState=E_Station.eReady,PT:=T#30S);
	IF tonMaxHeight.Q AND NOT bStateError  THEN
		bHeightMotorUp:=FALSE;
		bHeightMotorDown:=FALSE;
		bError := TRUE;
		udiErrorID:=7;
		udiErrorID := udiErrorID+iStationIndex;			
		sErrorDescription:='Wartość zadana wysokości jest większa od maksymalnej - zmień ustawienia w recepturze';
		sErrorDescription2:=REAL_TO_STRING(LREAL_TO_INT(lrMaxHeight));
	END_IF
	
	//Error 8 - ZBYT WYSOKA TEMPERATURA SILNIKA TYLNIEGO
	tonRearActualMotorTemperatureTooHigh(IN:=rRearActualMotorTemperature>130, PT:=T#10S);
	IF tonRearActualMotorTemperatureTooHigh.Q AND NOT bStateError THEN
		bHeightMotorUp:=FALSE;
		bHeightMotorDown:=FALSE;
		bStopped:=FALSE;
		bError := TRUE;
		udiErrorID	:=	8;
		udiErrorID	:=	udiErrorID+iStationIndex;
		sErrorDescription:='Zbyt wysoka temperatura napędu zakręcającego tylniego > 130C - zmniejsz moment zakręcania';
		sErrorDescription2:=INT_TO_STRING(REAL_TO_INT(rRearActualMotorTemperature));
	END_IF
	
	//Error 9 - ZBYT WYSOKA TEMPERATURA SILNIKA PRZEDNIEGO
	tonFrontActualMotorTemperatureTooHigh(IN:=rFrontActualMotorTemperature>130, PT:=T#10S);
	IF tonFrontActualMotorTemperatureTooHigh.Q AND NOT bStateError THEN
		bHeightMotorUp:=FALSE;
		bHeightMotorDown:=FALSE;
		bStopped:=FALSE;
		bError := TRUE;
		udiErrorID	:=	9;
		udiErrorID	:=	udiErrorID+iStationIndex;
		sErrorDescription:='Zbyt wysoka temperatura napędu zakręcającego przedniego > 130C - zmniejsz moment zakręcania';
		sErrorDescription2:=INT_TO_STRING(REAL_TO_INT(rFrontActualMotorTemperature));
	END_IF 	
ELSE
	bError := FALSE;	
END_IF

//******************PRZEJŚCIE DO eERROR*****************************

IF bError AND NOT bStateError THEN
	IF eLastState = eRunning THEN
		bCycleNotDone := TRUE;
	END_IF
	eState := E_Station.eError;
END_IF

//****************WYŚWIETLANIE STATUSU BLEDU***********************

(*Wyświetlanie błedu na wyjściu*)
bError;

(*Przepisywanie nazwy stacji*)
sErrorStationName := sStationName;
END_ACTION

ACTION HeightMotor:
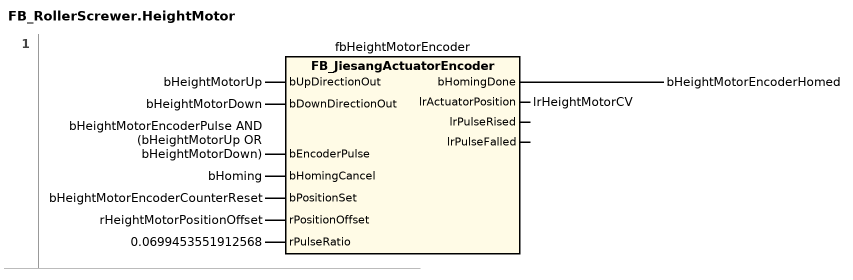
// NETWORK 1
fbHeightMotorEncoder(
    bUpDirectionOut := bHeightMotorUp,
    bDownDirectionOut := bHeightMotorDown,
    bEncoderPulse := bHeightMotorEncoderPulse AND (bHeightMotorUp OR bHeightMotorDown),
    bHomingCancel := bHoming,
    bPositionSet := bHeightMotorEncoderCounterReset,
    rPositionOffset := rHeightMotorPositionOffset,
    rPulseRatio := 0.0699453551912568,
    lrActuatorPosition => lrHeightMotorCV); // FB_JiesangActuatorEncoder
bHeightMotorEncoderHomed := fbHeightMotorEncoder.bHomingDone;
END_ACTION

ACTION Homing:
//BAZOWANIE
bPressingTopActuator:=FALSE;
bPressingRollsActuator:=FALSE;
	
//Podnoszenie stacji do maksymalnej pozycji
IF NOT bHeightMotorEncoderHomed OR rtEncoderHomed.Q THEN
	
	//Wylaczanie serwa zakręcania podczas bazowania
	mcScrewerFrontPower.Override:=100;
	mcScrewerFrontStop.Execute:=NOT bStopped;
	mcScrewerFrontMoveVelocity.Execute:=FALSE;
	mcScrewerFrontManualMove.JogBackwards:=FALSE;
	mcScrewerFrontManualMove.JogForward:=FALSE;
	
	mcScrewerRearPower.Override:=100;
	mcScrewerRearStop.Execute:=NOT bStopped;
	mcScrewerRearMoveVelocity.Execute:=FALSE;
	mcScrewerRearManualMove.JogBackwards:=FALSE;
	mcScrewerRearManualMove.JogForward:=FALSE;
	
	bHeightMotorUp:=TRUE;
	bHeightMotorDown:=FALSE;
	IF tonHeightNoChange.Q THEN
		bHeightMotorEncoderCounterReset:=TRUE;
		bHeightMotorUp:=FALSE;
    END_IF
	//Jesli enkoder zbazowany zakończ bazowanie	
	IF rtEncoderHomed.Q THEN
		bHeightMotorUp:=FALSE;
		bHeightMotorDown:=FALSE;
		eState:=E_Station.eHomingDone;
	END_IF		
		
//Po podniesieniu stacji opuszczanie do ustalonej wysokości
ELSIF bHeightMotorEncoderHomed THEN
	bHeightMotorEncoderCounterReset:=FALSE;
	bHeightMotorUp:=lrHeightMotorCV<=nPositionHeightSV;
	bHeightMotorDown:=lrHeightMotorCV>=nPositionHeightSV;
	//Kiedy stacja osiągnie wysokość zadaną
	IF ABS(lrHeightMotorCV-nPositionHeightSV)<1 OR tonLimitPosMaxReachedDelay.Q OR tonLimitPosMinReachedDelay.Q THEN
		bHeightMotorDown:=FALSE;
		bHeightMotorUp:=FALSE;
		eState:=E_Station.eHomingDone;
	END_IF			
END_IF
END_ACTION

ACTION ManualMovements:

//W trybie ruchów manualnych wykonuj ruchy za pomocą rozkazów manualnych
IF NOT bRun THEN
	mcScrewerFrontPower.Override:=lrManualOverride;
	uiScrewingFrontTorqueControl:=(INT_TO_UINT(iScrewerSetTorque+5)*10)*BOOL_TO_UINT(bManualScrewClockwise OR bManualScrewCClockwise);
	mcScrewerFrontManualMove.JogForward:=bManualScrewClockwise;	
	mcScrewerFrontManualMove.JogBackwards:=bManualScrewCClockwise;

	mcScrewerRearPower.Override:=lrManualOverride;
	uiScrewingRearTorqueControl:=(INT_TO_UINT(iScrewerSetTorque+5)*10)*BOOL_TO_UINT(bManualScrewClockwise OR bManualScrewCClockwise);
	mcScrewerRearManualMove.JogForward:=bManualScrewClockwise;	
	mcScrewerRearManualMove.JogBackwards:=bManualScrewCClockwise;
	
	bPressingTopActuator:=bManualPressingTopActuator;
	bPressingRollsActuator:=bManualPressingRollsActuator;
	bHeightMotorUp:=bManualHeightMotorUp;
	bHeightMotorDown:=bManualHeightMotorDown;
ELSE	//Kasuje zeby po cyklu nic sie nie poruszało
	bManualPressingTopActuator:=FALSE;
	bManualPressingRollsActuator:=FALSE;
	bManualHeightMotorUp  := FALSE;
	bManualHeightMotorDown  := FALSE;
END_IF


IF bHoming OR bHeightSet THEN
	eState:=E_Station.eHoming;
END_IF


Running();

	
//Zabezpieczenie przed kolizją stacji poprzez ruch podnośnika	
IF bHeightMotorDown AND lrHeightMotorCV<=lrMinHeight AND NOT bHoming AND NOT bHeightSet THEN
	bHeightMotorDown:=FALSE;
END_IF	

IF bHeightMotorUp AND lrHeightMotorCV>=lrMaxHeight AND NOT bHoming AND NOT bHeightSet THEN
	bHeightMotorUp:=FALSE;
END_IF		 

IF NOT bRun THEN
	bCycleDone 					:= FALSE;
	bCycleNotDone 				:= FALSE;
	bWarning					:= FALSE;		
END_IF
END_ACTION

ACTION Running:
//Timery
tofMotorUpPermition(IN:=bHeightMotorDown, PT:=T#250MS);
tofMotorDownPermition(IN:=bHeightMotorUp, PT:=T#250MS);	

CASE eRunningState OF

//====================================

	//Niegotowy
	E_RollerScrewer.eDisabled:
		eRunningState:=E_RollerScrewer.eReady;
	
	(*Oczekiwanie na wykonanie pojedynczego cyklu*)
	E_RollerScrewer.eReady:
        mcScrewerFrontSoftReset								(Axis:=RollerScrewerFrontAxisRef, Execute:=FALSE);                                       	
		mcScrewerFrontMoveVelocity.Execute					:=	FALSE;
		uiScrewingFrontTorqueControl						:=	6000; 
		
		mcScrewerRearSoftReset								(Axis:=RollerScrewerRearAxisRef, Execute:=FALSE);                                       	
		mcScrewerRearMoveVelocity.Execute					:=	FALSE;
		uiScrewingRearTorqueControl							:=	6000;    
		
		bScrewed											:=	FALSE;
		bScrewFound											:=	FALSE;
		tonTightScrewingTimer(IN:=FALSE,PT:=INT_TO_TIME(iScrewTightTime));                                           	
		IF NOT bCycleDone AND NOT bCycleNotDone THEN                                           	
			IF bRun THEN                	
				eRunningState							:=	E_RollerScrewer.ePushingCap;	
			END_IF
		END_IF


//====================================
	
		
	//ZAKRĘCARKA W STANIE WCISKANIA NAKRĘTKI
	E_RollerScrewer.ePushingCap:
			//ZRozkaz wciskania nakrętki od góry
			bPressingTopActuator:=nTopActuatorTimeDelayOff>0;
			//bPressingTopActuator:=TRUE;
			bPressingRollsActuator:=tonPushingCapDelay.Q; //zmiana1
			//Jeśli znikł czujnik wycofania docisku to przejdz dalej
			IF (NOT bUnPressedTopSensor OR nTopActuatorTimeDelayOff=0) AND bRollsPressedSensor AND tonRollsPressedDelay.Q THEN
				eRunningState:=E_RollerScrewer.ePushed;
			END_IF
			

		
//====================================		
				
	E_RollerScrewer.ePushed:
	
		IF bFindingScrewBeginingOption THEN
			mcScrewerFrontMoveRelative.Execute				:=	TRUE;
			mcScrewerFrontMoveRelative.Velocity				:=	lrScrewerSpeed;
			mcScrewerRearMoveRelative.Execute				:=	TRUE;
			mcScrewerRearMoveRelative.Velocity				:=	lrScrewerSpeed;			
			uiScrewingFrontTorqueControl						:=	4000;
			uiScrewingRearTorqueControl						:=	4000;
		END_IF
		mcScrewerFrontMoveVelocity.Velocity					:=	lrScrewerSpeed;
		mcScrewerRearMoveVelocity.Velocity					:=	lrScrewerSpeed;
		IF bFindingScrewBeginingOption THEN		
			eRunningState								:=	E_RollerScrewer.eFindingScrew;
			nMaxTorque									:=	0;
			nMinTorque									:=	2000;
			bScrewFound									:=	FALSE;	
		ELSE
			lrStartPositionScrewerFront					:=	RollerScrewerFrontAxisRef.NcToPlc.ActPos;
			lrStartPositionScrewerRear					:=	RollerScrewerRearAxisRef.NcToPlc.ActPos;
			eRunningState								:=	E_RollerScrewer.eScrewing;
			mcScrewerFrontMoveVelocity.Execute				:=	TRUE;
			mcScrewerRearMoveVelocity.Execute				:=	TRUE;
			lrStartScrewingPos							:=	RollerScrewerFrontAxisRef.NcToPlc.ActPos;		
		END_IF
			
	
//====================================					
	
	E_RollerScrewer.eFindingScrew:
	
			mcScrewerFrontMoveRelative.Execute				:=	TRUE;
			mcScrewerFrontMoveRelative.Velocity				:=	lrScrewerSpeed;
			mcScrewerRearMoveRelative.Execute				:=	TRUE;
			mcScrewerRearMoveRelative.Velocity				:=	lrScrewerSpeed;
			uiScrewingFrontTorqueControl					:=	4000;
			uiScrewingRearTorqueControl						:=	4000;	
			IF (mcScrewerFrontMoveRelative.Done AND mcScrewerRearMoveRelative.Done) OR bScrewFound THEN
			
				mcScrewerFrontMoveRelative.Execute			:=	FALSE;
				mcScrewerRearMoveRelative.Execute			:=	FALSE;
				bScrewFound									:=	TRUE;
				mcScrewerFrontHalt.Execute					:=	FALSE;
				mcScrewerRearHalt.Execute					:=	FALSE;	
				eRunningState								:=	E_RollerScrewer.eScrewing;
			
				mcScrewerFrontMoveVelocity.Execute			:=	TRUE;
				mcScrewerRearMoveVelocity.Execute			:=	TRUE;
				lrStartPositionScrewerFront					:=	RollerScrewerFrontAxisRef.NcToPlc.ActPos;
				lrStartPositionScrewerRear					:=	RollerScrewerRearAxisRef.NcToPlc.ActPos;
			END_IF	
			
	  			
//====================================				
		
	(*Zakręcanie*)
	E_RollerScrewer.eScrewing:
	
			mcScrewerFrontMoveVelocity.Velocity				:=	lrScrewerSpeed;
			mcScrewerRearMoveVelocity.Velocity				:=	lrScrewerSpeed;
			IF ABS(ABS(lrStartPositionScrewerFront)-ABS(RollerScrewerFrontAxisRef.NcToPlc.ActPos))>30 OR 
				ABS(ABS(lrStartPositionScrewerRear)-ABS(RollerScrewerRearAxisRef.NcToPlc.ActPos))>30
			THEN
				uiScrewingFrontTorqueControl					:=	INT_TO_UINT(iScrewerSetTorque+5)*10;
				uiScrewingRearTorqueControl						:=	INT_TO_UINT(iScrewerSetTorque+5)*10;
			ELSE
				uiScrewingFrontTorqueControl					:=	(INT_TO_UINT(iScrewerSetTorque+5)*10)+500;	
				uiScrewingRearTorqueControl						:=	(INT_TO_UINT(iScrewerSetTorque+5)*10)+500;
			END_IF
			mcScrewerFrontMoveVelocity.Direction				:=	MC_Direction.MC_Positive_Direction;
			mcScrewerRearMoveVelocity.Direction					:=	MC_Direction.MC_Positive_Direction;			
			IF tonTopActuatorDelayOff.Q THEN
				bPressingTopActuator					:=	FALSE; // Odcisniecie wczesniej niz zakręcanie
			END_IF
		
			IF tonTightScrewingTimer.Q THEN
				bPressingTopActuator					:=	FALSE;
				bPressingRollsActuator					:=	FALSE;
				mcScrewerFrontMoveVelocity.Execute			:=	FALSE;
				mcScrewerFrontSoftReset						(Axis:=RollerScrewerFrontAxisRef, Execute:= TRUE);
				mcScrewerRearMoveVelocity.Execute			:=	FALSE;
				mcScrewerRearSoftReset						(Axis:=RollerScrewerRearAxisRef, Execute:= TRUE);
				uiScrewingFrontTorqueControl					:=	0;
				uiScrewingRearTorqueControl					:=	0;			
				bScrewed								:=	TRUE;		
			END_IF
			IF tonPressingRollsReliseDelay.Q AND bScrewed THEN //200ms
				eRunningState							:=	E_RollerScrewer.eGoingUp;
			END_IF	
	

//====================================
						
	E_RollerScrewer.eGoingUp:
	
			mcScrewerFrontSoftReset							(Axis:=RollerScrewerFrontAxisRef, Execute:=TRUE);
			mcScrewerFrontStop.Execute						:=	FALSE;
			mcScrewerRearSoftReset							(Axis:=RollerScrewerRearAxisRef, Execute:=TRUE);
			mcScrewerRearStop.Execute						:=	FALSE;			
			IF bRollsUnPressedSensor AND bUnPressedTopSensor THEN
				eRunningState							:=	E_RollerScrewer.eDone;
			END_IF

	
//====================================	
		 
	E_RollerScrewer.eDone:
	
			bScrewed									:=	FALSE;
			bScrewFound									:=	FALSE;
			
			mcScrewerFrontSoftReset							(Axis:=RollerScrewerFrontAxisRef, Execute:=TRUE);
			mcScrewerFrontStop.Execute						:=	FALSE;
			mcScrewerRearSoftReset							(Axis:=RollerScrewerRearAxisRef, Execute:=TRUE);
			mcScrewerRearStop.Execute						:=	FALSE;
			uiScrewingFrontTorqueControl						:=	0;	
			uiScrewingRearTorqueControl						:=	0;				
			bCycleDone 									:= TRUE;
			eRunningState								:= E_RollerScrewer.eReady;
	

//====================================	
			
	E_RollerScrewer.eNotDone:
	
		bCycleNotDone 									:=	TRUE;
		eRunningState									:=	E_RollerScrewer.eReady;	
		mcScrewerFrontSoftReset								(Axis:=RollerScrewerFrontAxisRef, Execute:=TRUE);
		mcScrewerRearSoftReset								(Axis:=RollerScrewerRearAxisRef, Execute:=TRUE);	
	
END_CASE
END_ACTION

ACTION ServoFrontControlBlocks:
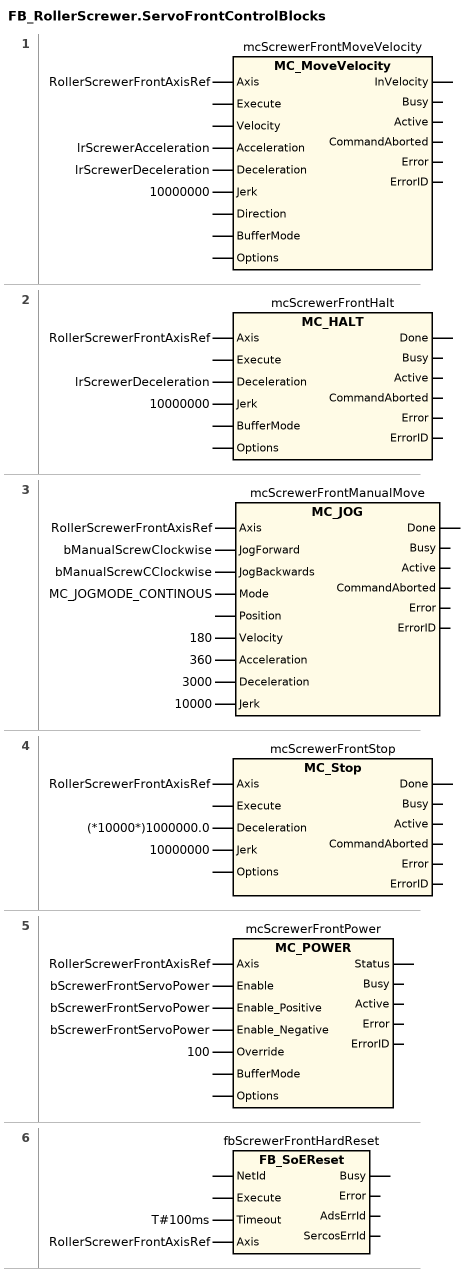
// NETWORK 1
mcScrewerFrontMoveVelocity(
    Axis := RollerScrewerFrontAxisRef,
    Acceleration := lrScrewerAcceleration,
    Deceleration := lrScrewerDeceleration,
    Jerk := 10000000); // MC_MoveVelocity

// NETWORK 2
mcScrewerFrontHalt(
    Axis := RollerScrewerFrontAxisRef,
    Deceleration := lrScrewerDeceleration,
    Jerk := 10000000); // MC_HALT

// NETWORK 3
mcScrewerFrontManualMove(
    Axis := RollerScrewerFrontAxisRef,
    JogForward := bManualScrewClockwise,
    JogBackwards := bManualScrewCClockwise,
    Mode := MC_JOGMODE_CONTINOUS,
    Velocity := 180,
    Acceleration := 360,
    Deceleration := 3000,
    Jerk := 10000); // MC_JOG

// NETWORK 4
mcScrewerFrontStop(Axis := RollerScrewerFrontAxisRef, Deceleration := (*10000*)1000000.0, Jerk := 10000000); // MC_Stop

// NETWORK 5
mcScrewerFrontPower(
    Axis := RollerScrewerFrontAxisRef,
    Enable := bScrewerFrontServoPower,
    Enable_Positive := bScrewerFrontServoPower,
    Enable_Negative := bScrewerFrontServoPower,
    Override := 100); // MC_POWER

// NETWORK 6
fbScrewerFrontHardReset(Timeout := T#100ms, Axis := RollerScrewerFrontAxisRef); // FB_SoEReset

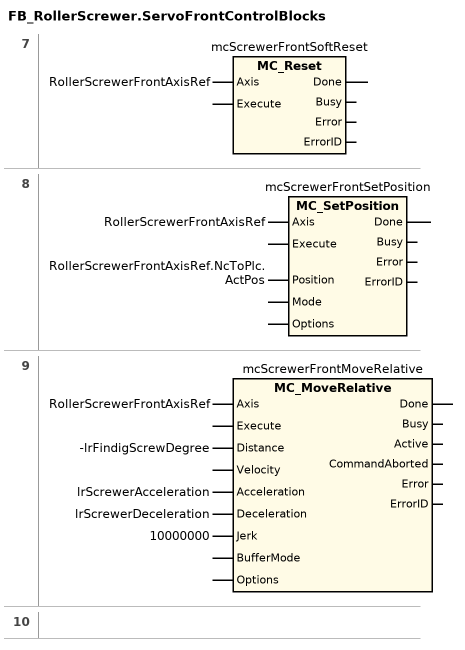
// NETWORK 7
mcScrewerFrontSoftReset(Axis := RollerScrewerFrontAxisRef); // MC_Reset

// NETWORK 8
mcScrewerFrontSetPosition(Axis := RollerScrewerFrontAxisRef, Position := RollerScrewerFrontAxisRef.NcToPlc.ActPos); // MC_SetPosition

// NETWORK 9
mcScrewerFrontMoveRelative(
    Axis := RollerScrewerFrontAxisRef,
    Distance := -lrFindigScrewDegree,
    Acceleration := lrScrewerAcceleration,
    Deceleration := lrScrewerDeceleration,
    Jerk := 10000000); // MC_MoveRelative

// NETWORK 10
END_ACTION

ACTION ServoRearControlBlocks:
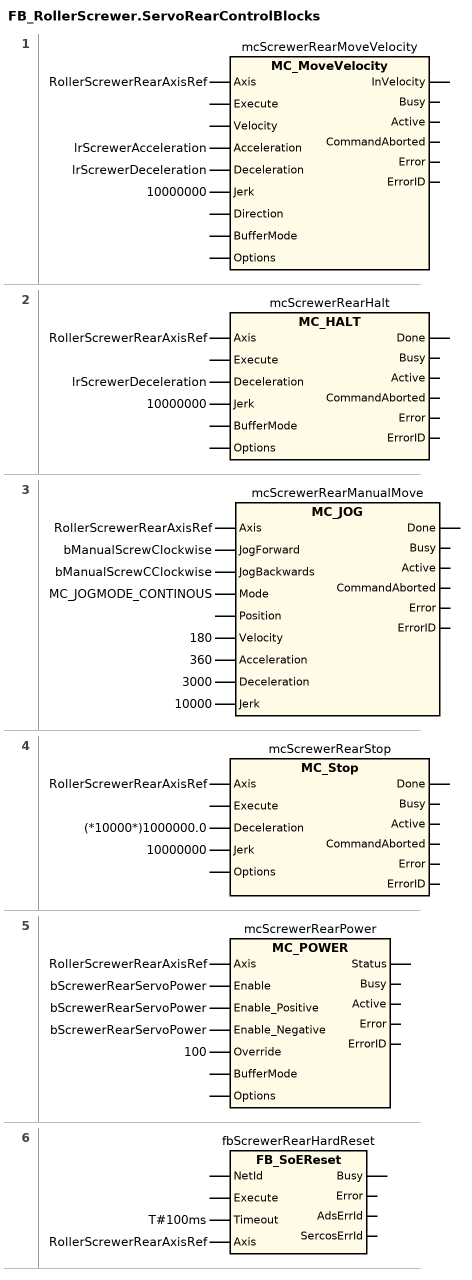
// NETWORK 1
mcScrewerRearMoveVelocity(
    Axis := RollerScrewerRearAxisRef,
    Acceleration := lrScrewerAcceleration,
    Deceleration := lrScrewerDeceleration,
    Jerk := 10000000); // MC_MoveVelocity

// NETWORK 2
mcScrewerRearHalt(Axis := RollerScrewerRearAxisRef, Deceleration := lrScrewerDeceleration, Jerk := 10000000); // MC_HALT

// NETWORK 3
mcScrewerRearManualMove(
    Axis := RollerScrewerRearAxisRef,
    JogForward := bManualScrewClockwise,
    JogBackwards := bManualScrewCClockwise,
    Mode := MC_JOGMODE_CONTINOUS,
    Velocity := 180,
    Acceleration := 360,
    Deceleration := 3000,
    Jerk := 10000); // MC_JOG

// NETWORK 4
mcScrewerRearStop(Axis := RollerScrewerRearAxisRef, Deceleration := (*10000*)1000000.0, Jerk := 10000000); // MC_Stop

// NETWORK 5
mcScrewerRearPower(
    Axis := RollerScrewerRearAxisRef,
    Enable := bScrewerRearServoPower,
    Enable_Positive := bScrewerRearServoPower,
    Enable_Negative := bScrewerRearServoPower,
    Override := 100); // MC_POWER

// NETWORK 6
fbScrewerRearHardReset(Timeout := T#100ms, Axis := RollerScrewerRearAxisRef); // FB_SoEReset

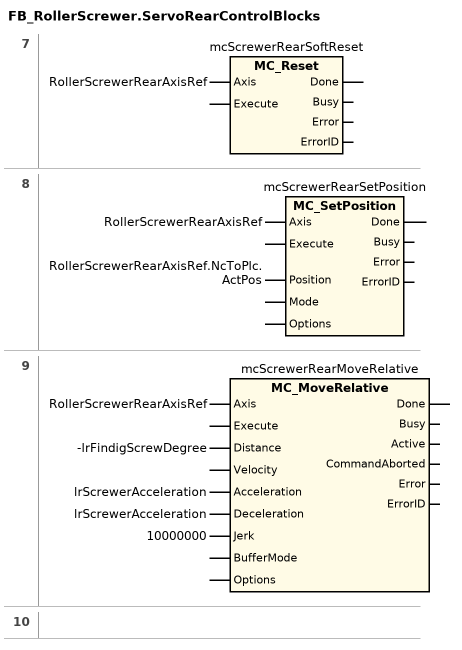
// NETWORK 7
mcScrewerRearSoftReset(Axis := RollerScrewerRearAxisRef); // MC_Reset

// NETWORK 8
mcScrewerRearSetPosition(Axis := RollerScrewerRearAxisRef, Position := RollerScrewerRearAxisRef.NcToPlc.ActPos); // MC_SetPosition

// NETWORK 9
mcScrewerRearMoveRelative(
    Axis := RollerScrewerRearAxisRef,
    Distance := -lrFindigScrewDegree,
    Acceleration := lrScrewerAcceleration,
    Deceleration := lrScrewerAcceleration,
    Jerk := 10000000); // MC_MoveRelative

// NETWORK 10
END_ACTION

ACTION Statistics:

rtrigCycleTimerRead(CLK:=(eRunningState=E_RollerScrewer.eDone) OR (eRunningState=E_RollerScrewer.eNotDone));
IF rtrigCycleTimerRead.Q THEN
	tCycleTime:=tonCycleTimer.ET;
END_IF
tonCycleTimer(IN:=eState>E_Station.eReady,PT:=T#1D);
END_ACTION

END_FUNCTION_BLOCK

// ---- POUs/FB/FB_JiesangActuatorEncoder.TcPOU
(*
Nazwa:			FB_JiesangActuatorEncoder
Opis:			Obsługa podnosnika Jiesang
Wersja:			v0.1
Data:			2018-10-10
Autor:			TW
Urzadzenia:		waga HBM
Konfiguracja:	
Info: 
- podlaczenie po RS485
*)

///!!!!!WAŻNE!!!!!!!!!!
///ABY ENKODER PRACOWAŁ POPRAWNIE TASK PLC MUSI BYĆ USTAWIONY NA 3ms!!!!!!!!!
///Wynika to z faktu że korzystamy ze zwykłych wejść cyfrowych a nie szybkich liczników!!!


FUNCTION_BLOCK FB_JiesangActuatorEncoder
VAR_INPUT
	bUpDirectionOut:BOOL;  	//Zmienna sterownika bezpośrednio sterująca siłownikiem w górę (zlinkowana z wyjściem sterownika)
	bDownDirectionOut:BOOL;	//Zmienna sterownika bezpośrednio sterująca siłownikiem w dół (zlinkowana z wyjsciem sterownika)
	bEncoderPulse:BOOL;		//Sygnał impulsów enkodera siłownika
	bHomingCancel:BOOL;		//Anulowanie bazowania enkodera
	bPositionSet:BOOL;		//Zmienna ustawia aktualną wartości pozycji zawartą w zmiennej 'nPositionOffset'
	rPositionOffset:REAL;		//Wartość do nadpisania aktualnej pozycji po ustawieniu wejścia 'AcbtorPositionSet'
	rPulseRatio:REAL;			//Przelicznik impulsów na mm  (pokonana_odleglosc_w_mm/ilość_impulsów)
	
	bOptionCoutingFalling : BOOL;  //Obliczenie spadania silnika
 END_VAR
VAR_OUTPUT
	bHomingDone:BOOL;
	lrActuatorPosition:LREAL:=-200;
	lrPulseRised:LREAL;
	lrPulseFalled:LREAL;
END_VAR
VAR
	tonOffDelay	:	TON;
rtEncoderPulse:R_TRIG;  //wykrywanie zbocza narastającego impulsu encodera
ftEncoderPulse:F_TRIG;  //wykrywanie zbocza opadającego impulsu encodera
rtActuatorPositionSet:R_TRIG;
bLastDirectionUp:BOOL;
rtHomingCancel: R_TRIG;
	cnt : INT;
END_VAR



//Kasowanie pozycjonowania enkodera
rtHomingCancel(CLK:=bHomingCancel,Q=>);
IF rtHomingCancel.Q THEN
	bHomingDone:=FALSE;
	lrActuatorPosition:=-200;
END_IF

//Jeśli na wejsciu pojawi sie ustawianie aktualnej pozycji enkodera
rtActuatorPositionSet(CLK:=bPositionSet,Q=>);
IF rtActuatorPositionSet.Q THEN
	lrActuatorPosition:=rPositionOffset;
	bHomingDone:=TRUE;
	lrPulseRised:=0;
	lrPulseFalled:=0;
END_IF


//Zapisywanie ostatniego kierunku ruchu siłownika
IF bUpDirectionOut AND NOT bDownDirectionOut THEN
	bLastDirectionUp:=TRUE;
ELSIF bDownDirectionOut AND NOT bUpDirectionOut THEN
	bLastDirectionUp:=FALSE;	
END_IF

//Wykrywanie zbocza pulsu enkodera
rtEncoderPulse(CLK:=bEncoderPulse,Q=>);
ftEncoderPulse(CLK:=bEncoderPulse,Q=>);

tonOffDelay(IN:= NOT bUpDirectionOut AND NOT bDownDirectionOut, PT:=T#2S);

IF NOT bOptionCoutingFalling THEN
	IF rtEncoderPulse.Q OR ftEncoderPulse.Q THEN
		IF bLastDirectionUp THEN
			lrActuatorPosition:=lrActuatorPosition+rPulseRatio;
		ELSE
			lrActuatorPosition:=lrActuatorPosition-rPulseRatio;
		END_IF	
	END_IF
ELSE
	IF (bUpDirectionOut OR bDownDirectionOut) THEN
		IF rtEncoderPulse.Q OR ftEncoderPulse.Q THEN
			IF bLastDirectionUp THEN
				lrActuatorPosition:=lrActuatorPosition+rPulseRatio;
			ELSE
				lrActuatorPosition:=lrActuatorPosition-rPulseRatio;
			END_IF	
		END_IF
	ELSIF (NOT tonOffDelay.Q AND (rtEncoderPulse.Q OR ftEncoderPulse.Q)) THEN
		lrActuatorPosition:=lrActuatorPosition-rPulseRatio;
		cnt:=cnt +1;
	END_IF	
END_IF

END_FUNCTION_BLOCK

// ---- POUs/P02_BottlePusher.TcPOU
(*
Nazwa:			P02_BottlePusher
Opis:			Stacja wbijaka butelek
Wersja:			v0.1
Data:			2024-05-21
Autor:			DP
Urzadzenia:		
Konfiguracja:	
Info:
*)

PROGRAM P02_BottlePusher
VAR
	
	fbBottlePusher									:FB_Gate;
	eBottlePusherState								:E_Station; 									
	eBottlePusherRunningState						:E_Barrier; 
	fbBottlePusherState								:FB_State;	

	QbBottlePusherActuator 							:BOOL;
	IbBottlePusherActuatorSensor 			AT %I*  :BOOL; 
	IbBottlePusherBottleBeforeSensor 		AT %I*  :BOOL; 
	IbBottlePusherBottleAfterSensor 		AT %I*  :BOOL;

	
	tonfbBottlePusherDownSensor						:TON;
END_VAR

aBottlePusher();


tonfbBottlePusherDownSensor	(IN:= QbBottlePusherActuator, PT:=T#500MS);

ACTION aBottlePusher:
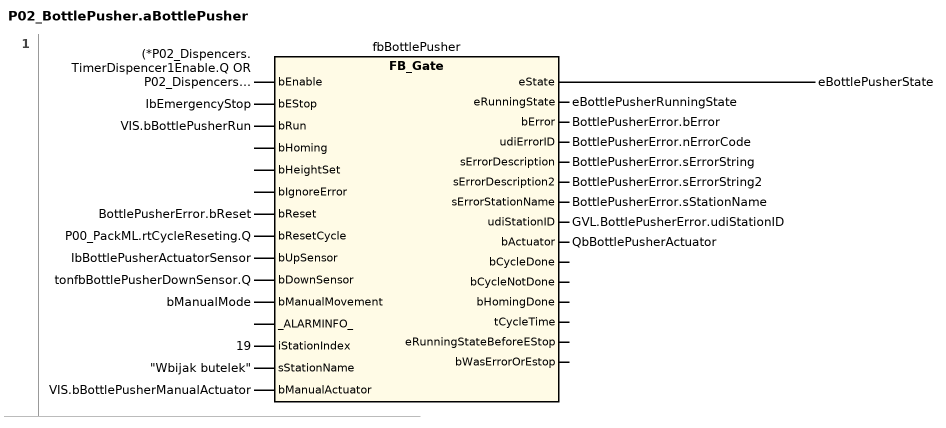
// NETWORK 1
fbBottlePusher(
    bEnable := (*P02_Dispencers.TimerDispencer1Enable.Q OR P02_Dispencers.TimerDispencer3Enable.Q*)FALSE,
    bEStop := IbEmergencyStop,
    bRun := VIS.bBottlePusherRun,
    bReset := BottlePusherError.bReset,
    bResetCycle := P00_PackML.rtCycleReseting.Q,
    bUpSensor := IbBottlePusherActuatorSensor,
    bDownSensor := tonfbBottlePusherDownSensor.Q,
    bManualMovement := bManualMode,
    iStationIndex := 19,
    sStationName := "Wbijak butelek",
    bManualActuator := VIS.bBottlePusherManualActuator,
    eRunningState => eBottlePusherRunningState,
    bError => BottlePusherError.bError,
    udiErrorID => BottlePusherError.nErrorCode,
    sErrorDescription => BottlePusherError.sErrorString,
    sErrorDescription2 => BottlePusherError.sErrorString2,
    sErrorStationName => BottlePusherError.sStationName,
    udiStationID => GVL.BottlePusherError.udiStationID,
    bActuator => QbBottlePusherActuator); // FB_Gate
eBottlePusherState := fbBottlePusher.eState;
END_ACTION

END_PROGRAM

// ---- POUs/P13_BottleTransferAfterDrag.TcPOU
(*
Nazwa:			P13_BottleTransferAfterDrag
Opis:			Stacja przesuwania formatek za robotem
Wersja:			v0.1
Data:			2025-12-22
Autor:			DP
Urzadzenia:		
Konfiguracja:	
Info:

*)
PROGRAM P13_BottleTransferAfterDrag
VAR
	
	(*DI wyspy pneumatycznej*)
	QABPneumatic648ValveCoils 							AT %Q* 	: ARRAY[1..5] OF BYTE;	
	IABPneumatic648DigitalInput 						AT %I* 	: ARRAY[1..4] OF BYTE;
	IuiPneumatic648State								AT %I* 	: UINT;	
	                                                	
	(*******PRZECIAGANIE**********)                 	
	fbBottleTransferAfterDrag							: FB_FormsDragActuator;
	eBottleTransferAfterDragState						: E_Station;					
	eBottleTransferAfterDragRunningState				: E_DragStationState;			
	fbBottleTransferAfterDragState						: FB_State;
	
	//WEJSCIA I WYJSCIA SPRZETOW

	IbBottleTransferAfterDragOnSensor 					: BOOL;			// Czujnik 
	IbBottleTransferAfterDragOffSensor 					: BOOL;			// Czujnik 	
	IbBottleTransferAfterDragStoperOnSensor 			: BOOL;			// Czujnik 	
	IbBottleTransferAfterDragGateOnSensor 				: BOOL;			// Czujnik 		
	IbBottleTransferAfterDragFirstFormSensor 			: BOOL;			// Czujnik
	IbBottleTransferAfterDragSecondFormSensor	 		: BOOL;			// Czujnik
	IbBottleTransferAfterDragAfterSensor 				: BOOL;			// Czujnik

	bTemp:BOOL;
END_VAR

a5_Draging();
aPneumatics();

ACTION a5_Draging:
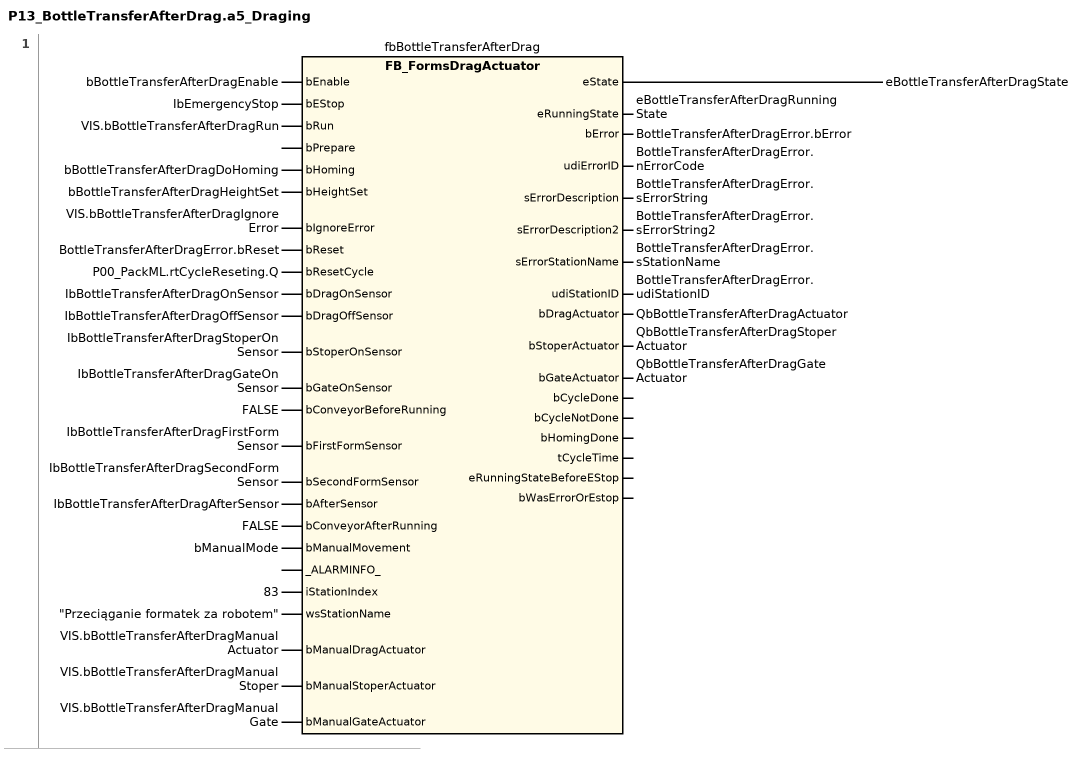
// NETWORK 1
fbBottleTransferAfterDrag(
    bEnable := bBottleTransferAfterDragEnable,
    bEStop := IbEmergencyStop,
    bRun := VIS.bBottleTransferAfterDragRun,
    bHoming := bBottleTransferAfterDragDoHoming,
    bHeightSet := bBottleTransferAfterDragHeightSet,
    bIgnoreError := VIS.bBottleTransferAfterDragIgnoreError,
    bReset := BottleTransferAfterDragError.bReset,
    bResetCycle := P00_PackML.rtCycleReseting.Q,
    bDragOnSensor := IbBottleTransferAfterDragOnSensor,
    bDragOffSensor := IbBottleTransferAfterDragOffSensor,
    bStoperOnSensor := IbBottleTransferAfterDragStoperOnSensor,
    bGateOnSensor := IbBottleTransferAfterDragGateOnSensor,
    bConveyorBeforeRunning := FALSE,
    bFirstFormSensor := IbBottleTransferAfterDragFirstFormSensor,
    bSecondFormSensor := IbBottleTransferAfterDragSecondFormSensor,
    bAfterSensor := IbBottleTransferAfterDragAfterSensor,
    bConveyorAfterRunning := FALSE,
    bManualMovement := bManualMode,
    iStationIndex := 83,
    wsStationName := "Przeciąganie formatek za robotem",
    bManualDragActuator := VIS.bBottleTransferAfterDragManualActuator,
    bManualStoperActuator := VIS.bBottleTransferAfterDragManualStoper,
    bManualGateActuator := VIS.bBottleTransferAfterDragManualGate,
    eRunningState => eBottleTransferAfterDragRunningState,
    bError => BottleTransferAfterDragError.bError,
    udiErrorID => BottleTransferAfterDragError.nErrorCode,
    sErrorDescription => BottleTransferAfterDragError.sErrorString,
    sErrorDescription2 => BottleTransferAfterDragError.sErrorString2,
    sErrorStationName => BottleTransferAfterDragError.sStationName,
    udiStationID => BottleTransferAfterDragError.udiStationID,
    bDragActuator => QbBottleTransferAfterDragActuator,
    bStoperActuator => QbBottleTransferAfterDragStoperActuator,
    bGateActuator => QbBottleTransferAfterDragGateActuator); // FB_FormsDragActuator
eBottleTransferAfterDragState := fbBottleTransferAfterDrag.eState;
END_ACTION

ACTION aPneumatics:
// Do podpięcia według kolejności
QbBottleTransferAfterDragActuator		;
QbBottleTransferAfterDragStoperActuator	;
QbBottleTransferAfterDragGateActuator	;

(*************************** EB1 **************************************)
// Wyspa 1 - przeciaganie za rrobotem
IuiPneumatic648State;
QABPneumatic648ValveCoils[1].0	:= QbBottleTransferAfterDragActuator;
QABPneumatic648ValveCoils[1].1 	:= NOT  QbBottleTransferAfterDragActuator;               
QABPneumatic648ValveCoils[1].2 	:=  QbBottleTransferAfterDragStoperActuator;
QABPneumatic648ValveCoils[1].3 	:= NOT QbBottleTransferAfterDragStoperActuator;                   	                    
QABPneumatic648ValveCoils[1].4 	:=  QbBottleTransferAfterDragGateActuator;
QABPneumatic648ValveCoils[1].5 	:= NOT QbBottleTransferAfterDragGateActuator;
QABPneumatic648ValveCoils[1].6 	;
QABPneumatic648ValveCoils[1].7 	;
QABPneumatic648ValveCoils[2].0 	;
QABPneumatic648ValveCoils[2].1  ;
QABPneumatic648ValveCoils[2].2 	;
QABPneumatic648ValveCoils[2].3 	;
QABPneumatic648ValveCoils[2].4 	;		
QABPneumatic648ValveCoils[2].5 	;
QABPneumatic648ValveCoils[2].6 	;
QABPneumatic648ValveCoils[2].7 	;
                                                      
(*********************Koniec ROPP EB1 **************************************) 

//Zawór głównego powietrza
//QbROPPCompressedAir	:=	IbEmergencyStop;

(*************************** 648 EB1 **************************************)
// Wyspa 1 - 52N8
IuiPneumatic648State;
//DI1

IbBottleTransferAfterDragOffSensor 			:=		IABPneumatic648DigitalInput[1].0;	
IbBottleTransferAfterDragOnSensor 			:=		IABPneumatic648DigitalInput[1].1;	
IbBottleTransferAfterDragStoperOnSensor 	:=		IABPneumatic648DigitalInput[1].2;
IbBottleTransferAfterDragGateOnSensor 		:=		IABPneumatic648DigitalInput[1].3;   
IbBottleTransferAfterDragFirstFormSensor 	:=		IABPneumatic648DigitalInput[1].4;	
IbBottleTransferAfterDragSecondFormSensor	:=		IABPneumatic648DigitalInput[1].5;	
IbBottleTransferAfterDragAfterSensor 		:=		IABPneumatic648DigitalInput[1].6;	
IABPneumatic648DigitalInput[1].7;	
                                    
IABPneumatic648DigitalInput[2].0;	
IABPneumatic648DigitalInput[2].1;	
IABPneumatic648DigitalInput[2].2;	
IABPneumatic648DigitalInput[2].3;
IABPneumatic648DigitalInput[2].4;	
IABPneumatic648DigitalInput[2].5;		
IABPneumatic648DigitalInput[2].6;		
IABPneumatic648DigitalInput[2].7;	

(*********************Koniec 648 **************************************)
END_ACTION

END_PROGRAM

// ---- POUs/FB/NewFBs/FB_FormsDragActuator.TcPOU
(*
Nazwa:		FB_FormsDragActuator
Opis:		Przeciąganie formatek 
Wersja:		V0.5
Data:		2025-12-22
Autor:		DJ, DP
Urządzenia:	Siłownik podnoszenia wideł, Silnik krokowy przeciągania 
Ostatnie zmiany:
	- 20250904 [DP] EventLog->wywołać błędy 
	- 2025-08-19 [DP] Homing false
	- 2024-11-25 [DP] Czujnik dół
	- 2024-10-01 [DP] ESTOP Delay
	- RRRR-MM-DD [KTO?] Tekst Tekst Tekst Tekst Tekst Tekst Tekst Tekst Tekst Tekst 
	- 2025-09-15[VS] Jazda i stop w pozycji końcowej
Konfiguracja:
	- Krokówka
	Instukcja:
		-
		-
		-
	
Info:
	- Obsługa tylko jednego siłownika podnoszenia i dwóch siłowników prowadzących

*)

FUNCTION_BLOCK FB_FormsDragActuator
VAR_INPUT
	bEnable										: BOOL;				//Zezwolenie na pracę
	bEStop										: BOOL;				//Stop awaryjny włączony
	bRun										: BOOL;				//Rozkaz przeciagania
	bPrepare									: BOOL;				//Rozkaz przygotownaia 
	bHoming										: BOOL;				//Zezwolenie na wykonanie bazowania i pozycjonowanie układu
	bHeightSet									: BOOL;				//Ustaw do pozycji
	bIgnoreError								: BOOL;				//Ignorowanie błędów 
	bReset										: BOOL;				//Reset błędu, jeśli jest w stanie "eError"
	bResetCycle									: BOOL;				//Reset cyklu


	bDragOnSensor								: BOOL;				//
	bDragOffSensor								: BOOL;				//
	bStoperOnSensor								: BOOL;				//
	bGateOnSensor								: BOOL;				//

	bConveyorBeforeRunning						: BOOL;	
	bFirstFormSensor							: BOOL;
	bSecondFormSensor							: BOOL;
	bAfterSensor								: BOOL;	
	bConveyorAfterRunning						: BOOL;		
	
	bManualMovement								: BOOL;				//Zezwolenie na ruchy ręczne

	_ALARMINFO_									: BOOL;
	iStationIndex								: UDINT;
	wsStationName								: WSTRING;
END_VAR

VAR_OUTPUT
	eState										: E_Station;
	eRunningState								: E_DragStationState;	// Stan przeciągania formatek
	bError										: BOOL;					// Błąd stacji
	udiErrorID									: UDINT;				// Nr blędu przeciągania formatek
	sErrorDescription							: STRING(200);			// Opis błędu
	sErrorDescription2							: STRING(200);			// Opis błędu
	sErrorStationName							: STRING;				// Nazwa stacji
	udiStationID								: UDINT;				// Nr stacji

	bDragActuator								: BOOL;					
	bStoperActuator								: BOOL;					
	bGateActuator								: BOOL;					
	
	bCycleDone									: BOOL;					//Sygnał zakończenia cyklu
	bCycleNotDone								: BOOL;
	bHomingDone									: BOOL;
	tCycleTime									: TIME;					//Czas cyklu
	//Dodatkowe	
	eRunningStateBeforeEStop					: E_DragStationState;	//Stan przed E-Stopem	
	bWasErrorOrEstop							: BOOL;
	
END_VAR

VAR
	(*LastStates*)
	eLastState									: E_Station;						//Stan ogólny bloku
	eLastStateTemp								: E_Station;						//Stan ogólny bloku
	eLastRunningState							: E_DragStationState;				//Stan podbloku
	eLastRunningStateTemp						: E_DragStationState;				//Stan podbloku
		                                    		                                 		
	(*Control*)
	tonResetting								: TON;								//Czas resetu
	tonHoming									: TON;
	tonPreparingToReady							: TON;								//Czas potrzeby na przygotowanie osi
	rtResetCommands								: R_TRIG;                                    	
	rtResetCycle								: R_TRIG;

	(*Statistics*)
	tonCycleTimer								: TON;								//Czas cyklu przeciągania	
	rtrigCycleTimerRead							: R_TRIG;

	(*Homing*)
	iHomingCase									: INT;
	
	(*Aborting*)
	iAbortingCase								: INT;
	                                    	
	(*Errors*)
	bStateError									: BOOL;
	tonEstopDelay								: TON;
	bResetCycleOn								: BOOL;
	tonbDragOnSensor							: TON;	
	tonbDragOffSensor							: TON;		
	tonbStoperOnSensor							: TON;
	tonbGateSensor								: TON;
	tonBeforeSensor								: TON;	
	tonAfterSensor								: TON;
		
	(*Running*)
	tonNotDragActuatorDelay						: TON;
	tonRunningDraging							: TON;
	tonRunningLifting							: TON;
	tonRunningeEndingOfDrag						: TON;
	(*Inne*)
	
	//Zmienne od EVENTLOGGER
	bAlarmInit 						: BOOL := TRUE; 
	nAlarmNumerator					: INT;
	arfbAlarm						: ARRAY[0..19] OF  FB_TcAlarm;		//Tablica bloczków błędów
	fbSourceInfo 					: FB_TcSourceInfo;
	iSourceInfo						: I_TcSourceInfo;
	sAlarmTest						: STRING;
	//Koniec zmiennych od EVENTLOGGER
	
END_VAR
	
VAR_IN_OUT
	bManualDragActuator							: BOOL;		
	bManualStoperActuator						: BOOL;			
	bManualGateActuator							: BOOL;			
END_VAR

ResetAll();
ErrorHandling();
Signals();
Control();
Limits();
Statistics();
aStationID();
(*Zapisywanie ostatniego stanu*)
IF eLastStateTemp<>eState THEN
	eLastState := eLastStateTemp;
END_IF
eLastStateTemp := eState;
IF eLastRunningStateTemp<>eRunningState THEN
	eLastRunningState := eLastRunningStateTemp;
END_IF
eLastRunningStateTemp := eRunningState;
(*Koniec Zapisywanie ostatniego stanu*)

ACTION aStationID:
udiStationID	:=	iStationIndex;
END_ACTION

ACTION Control:


	(*****Wyłączenie enable*****)
	IF NOT bEnable AND NOT bError THEN
		IF eState <> E_Station.eDisabled AND eState <> E_Station.ePreparingToDisable THEN
				eState 								:= E_Station.ePreparingToDisable; 
		END_IF	
	END_IF

	(*****Estop*****)
	IF NOT bEstop  THEN	
		IF eState <> E_Station.eAborted AND eState <> E_Station.eAborting AND eState <> E_Station.eDisabled THEN
				eRunningStateBeforeEStop			:= eRunningState;
				eState 								:= E_Station.eAborting; 
				iAbortingCase						:= 0; 
		END_IF
	END_IF


	
CASE eState OF
	
//==========================================================================================	
	E_Station.eDisabled: 						// Stan nieaktywnosci (Stacja wyłączona) 
		
		IF bEnable THEN
			eState 									:= E_Station.ePreparingToReady; 
		END_IF 

//==========================================================================================	    
	E_Station.eAborted: 						// Stan bezpiecznego zatrzymania (po Abortingu) 	
			
		IF bEStop THEN
			bWasErrorOrEstop						:= TRUE;	
			eState 									:= E_Station.ePreparingToReady;
		END_IF		
			
//==========================================================================================	
	E_Station.eAborting:                 		// Stan bezpiecznego zatrzymywania (po EStopie)
		
		CASE iAbortingCase OF
			
			0: //Inicjalizacja
				iAbortingCase						:= 40;
				
			40: //Kasowanie podzespołow
				ResetCommands();
				iAbortingCase						:= 50;
				
			50: //Przejście do Aborted
				iAbortingCase						:= 0;
				eState								:= E_Station.eAborted;
				eRunningState						:= E_DragStationState.eReady;
				
		END_CASE

//==========================================================================================			
	E_Station.eError:                 	 		// Stan błędu 	
		
		bWasErrorOrEstop							:= TRUE;

		IF bReset THEN
			eState									:= E_Station.eResetting;	
		ELSE
			ResetCommands();
		END_IF
			
//==========================================================================================
	E_Station.eResetting:						// Stan resetowania bledu (po Errorze)
			
		IF  		arfbAlarm[0].bActive OR arfbAlarm[1].bActive OR arfbAlarm[2].bActive 
			 	OR	arfbAlarm[3].bActive OR arfbAlarm[4].bActive OR arfbAlarm[4].bActive  
		THEN
			bDragActuator								:=	FALSE;	
			bStoperActuator								:=	TRUE;	
			bGateActuator								:=	FALSE;		
			bError										:=	FALSE;
		END_IF	
	
		IF NOT bError THEN
			udiErrorID									:= 0;
			sErrorDescription							:= '';
			sErrorDescription2							:= '';	
			eState										:= E_Station.ePreparingToReady;
		ELSIF tonResetting.Q THEN                   	
			eState										:= E_Station.eError;
		END_IF	
 
//==========================================================================================
	E_Station.eManualMovement:     				// Stan ruchów manualnych  
       
		ManualMovements();
		//Wyjście z trybu serwisowego
		IF NOT bManualMovement THEN
			bDragActuator							:=	bManualDragActuator;	
			bStoperActuator							:=	bManualStoperActuator;
			bGateActuator							:=	bManualGateActuator;
			eState									:=	E_Station.eReady;
		END_IF 

//==========================================================================================		
	E_Station.eHoming:							// Stan bazowania 
		
		Homing();	
		IF NOT bHoming AND NOT bHeightSet AND tonHoming.Q THEN
			eState									:=	E_Station.ePreparingToReady;
		END_IF		
			
//==========================================================================================
	E_Station.eHomingDone:                  	// Stan wykonania bazowania 

		bHomingDone									:= TRUE;
		bResetCycleOn								:= FALSE;		
		IF NOT bHoming AND NOT bHeightSet AND NOT bResetCycleOn THEN
			eState									:=	E_Station.ePreparingToReady;
		END_IF

//==========================================================================================
	E_Station.ePreparingToReady:            	// Stan przygotowywania do gotowosci (zawsze przed Ready)  

		IF tonPreparingToReady.Q THEN
						
				ResetCommands();
				eState								:= E_Station.eReady;
				eRunningState						:= E_DragStationState.eReady;
				IF bResetCycleOn THEN
					eState							:= E_Station.eHoming;
				END_IF
		
		END_IF			

//==========================================================================================
	E_Station.ePreparingToDisable:         	 	// Stan przygotowywania do nieaktywnosci (po wyłączeniu Enable) 
  

		bWasErrorOrEstop							:= FALSE;
		bHomingDone									:= FALSE;	
		
		ResetCommands();
		eState									:= 	E_Station.eDisabled;
		eRunningState							:= 	E_DragStationState.eReady;
		

//==========================================================================================	
	E_Station.eReady:							// Stan gotowosci 


		(*Skasowanie wszystkich komend*)
		IF rtResetCommands.Q THEN	ResetCommands();	END_IF		
		
	
		IF (bRun OR bPrepare) AND NOT bCycleDone THEN
			eState									:= E_Station.eStarting;		
		END_IF		
		IF bHoming OR bHeightSet THEN
			eState									:= E_Station.eHoming;
		END_IF
		IF bManualMovement THEN
			bManualDragActuator						:=	bDragActuator;			
			bManualStoperActuator					:=	bStoperActuator;	
			bManualGateActuator						:=	bGateActuator;	
			eState									:=	E_Station.eManualMovement;					
		END_IF
		IF NOT bRun AND NOT bPrepare THEN
			bCycleDone								:= FALSE;
		END_IF

//==========================================================================================
	E_Station.eStopping:					// Stan zatrzymywania 
		
		Running();
		eState 									:= E_Station.eReady;

//==========================================================================================
	E_Station.eStarting:                  	// Stan uruchamiania (po Ready)
		
		eState										:= E_Station.eRunning;

//==========================================================================================
	E_Station.eRunning:               		// Stan wykonywania cyklu (po Startingu), w tym stanie osobny
 
		Running();

		IF NOT bRun AND NOT bPrepare THEN					(*Przerywanie cyklu*)
			eState 				 					:= E_Station.eStopping;	
		END_IF
			
		IF bCycleDone THEN (*Cykl zakończony*)
			eState 				 					:= E_Station.eReady;
		END_IF	
		
//==========================================================================================
END_CASE
END_ACTION

ACTION ErrorHandling:
// Alarm_0610	610	Error	Siłownik przeciągania | Blokada wysunięcia - sprawdź czujnik lub odblokuj  
// Alarm_0611	611	Error	Siłownik przeciągania | Blokada wsunięcia - sprawdź czujnik lub odblokuj  
// Alarm_0612	612	Error	Banda końcowa | Blokada wysunięcia - sprawdź czujnik lub odblokuj  
// Alarm_0613	613	Error	Szlaban | Blokada wysunięcia - sprawdź czujnik lub odblokuj  
// Alarm_0614	614	Error	Bład czujników przed przeciąganiem - sprawdź ułożenie formatek
// Alarm_0615	615	Error	Bład czujników za przeciąganiem - sprawdź ułożenie formatek

